SPLINE
SPL {X  -162.820, Y  +428.091, Z    +0.000, E1   +59.583, E3 +218892.152}
SPL {X  -162.820, Y  +410.436, Z    +0.000, E1   +60.611, E3 +218906.354}
SPL {X  -162.820, Y  +392.633, Z    +0.000, E1   +61.698, E3 +218919.086}
SPL {X  -162.753, Y  +375.814, Z    +0.000, E1   +62.427, E3 +218932.608}
SPL {X  -161.572, Y  +360.382, Z    +0.000, E1   +62.315, E3 +218950.211}
SPL {X  -160.005, Y  +350.357, Z    +0.000, E1   +62.043, E3 +218962.774}
SPL {X  -158.606, Y  +343.697, Z    +0.000, E1   +61.897, E3 +218970.997}
SPL {X  -156.311, Y  +334.925, Z    +0.000, E1   +61.505, E3 +218983.343}
SPL {X  -153.198, Y  +325.358, Z    +0.000, E1   +61.117, E3 +218996.036}
SPL {X  -151.022, Y  +319.651, Z    +0.000, E1   +60.776, E3 +219004.208}
SPL {X  -149.105, Y  +315.094, Z    +0.000, E1   +60.301, E3 +219011.961}
SPL {X  -146.196, Y  +308.826, Z    +0.000, E1   +59.961, E3 +219020.668}
SPL {X  -143.704, Y  +303.952, Z    +0.000, E1   +59.374, E3 +219029.025}
SPL {X  -140.940, Y  +298.976, Z    +0.000, E1   +59.075, E3 +219035.950}
SPL {X  -137.763, Y  +293.715, Z    +0.000, E1   +58.761, E3 +219043.057}
SPL {X  -129.725, Y  +282.103, Z    +0.000, E1   +61.069, E3 +219044.560}
SPL {X  -106.695, Y  +257.510, Z    +0.000, E1   +52.408, E3 +219145.282}
SPL {X  -104.122, Y  +255.325, Z    +0.000, E1   +51.312, E3 +219235.340}
ENDSPLINE

SPLINE
SPL {X  -140.007, Y  +297.383, Z    +0.000, E1   +42.766, E3 +219274.665}
SPL {X  -156.919, Y  +337.064, Z    +0.000, E1   +27.647, E3 +219280.816}
SPL {X  -160.736, Y  +354.534, Z    +0.000, E1   +18.553, E3 +219283.511}
SPL {X  -162.078, Y  +364.978, Z    +0.000, E1   +12.369, E3 +219285.196}
SPL {X  -162.656, Y  +373.196, Z    +0.000, E1    +6.960, E3 +219284.692}
SPL {X  -162.819, Y  +379.805, Z    +0.000, E1    +2.285, E3 +219284.816}
SPL {X  -162.820, Y  +382.797, Z    +0.000, E1    -0.206, E3 +219284.322}
SPL {X  -162.820, Y  +386.214, Z    +0.000, E1    -4.241, E3 +219284.088}
SPL {X  -162.820, Y  +390.506, Z    +0.000, E1   -10.770, E3 +219283.854}
SPL {X  -162.820, Y  +394.643, Z    +0.000, E1   -17.317, E3 +219283.808}
SPL {X  -162.820, Y  +401.515, Z    +0.000, E1   -27.960, E3 +219284.628}
SPL {X  -162.820, Y  +412.105, Z    +0.000, E1   -42.847, E3 +219283.620}
SPL {X  -162.820, Y  +422.796, Z    +0.000, E1   -52.392, E3 +219284.841}
SPL {X  -162.820, Y  +474.423, Z    +0.000, E1   -65.078, E3 +219305.892}
SPL {X  -162.820, Y  +578.686, Z    +0.000, E1   -67.085, E3 +219375.056}
ENDSPLINE

SPLINE
SPL {X  -162.820, Y  +565.364, Z    +0.000, E1   -63.589, E3 +219389.056}
ENDSPLINE

SPLINE
SPL {X  -162.820, Y  +574.608, Z    +0.000, E1   -63.370, E3 +219400.315}
SPL {X  -162.820, Y  +584.314, Z    +0.000, E1   -63.342, E3 +219410.607}
SPL {X  -162.820, Y  +593.857, Z    +0.000, E1   -63.382, E3 +219420.310}
SPL {X  -162.820, Y  +602.272, Z    +0.000, E1   -63.279, E3 +219429.838}
SPL {X  -162.820, Y  +613.309, Z    +0.000, E1   -63.489, E3 +219439.836}
SPL {X  -162.820, Y  +627.013, Z    +0.000, E1   -63.389, E3 +219455.057}
SPL {X  -162.820, Y  +642.772, Z    +0.000, E1   -63.348, E3 +219471.716}
SPL {X  -162.820, Y  +651.969, Z    +0.000, E1   -63.137, E3 +219482.778}
SPL {X  -162.820, Y  +662.662, Z    +0.000, E1   -63.383, E3 +219492.236}
SPL {X  -162.819, Y  +673.983, Z    +0.000, E1   -63.398, E3 +219503.958}
SPL {X  -162.399, Y  +685.202, Z    +0.000, E1   -63.235, E3 +219516.952}
SPL {X  -161.289, Y  +695.772, Z    +0.000, E1   -63.167, E3 +219528.402}
SPL {X  -160.212, Y  +702.527, Z    +0.000, E1   -62.898, E3 +219537.383}
SPL {X  -158.647, Y  +710.128, Z    +0.000, E1   -62.776, E3 +219546.206}
SPL {X  -156.957, Y  +716.799, Z    +0.000, E1   -62.460, E3 +219555.324}
SPL {X  -155.130, Y  +722.947, Z    +0.000, E1   -62.207, E3 +219563.436}
SPL {X  -152.287, Y  +731.112, Z    +0.000, E1   -61.798, E3 +219574.711}
SPL {X  -149.420, Y  +738.185, Z    +0.000, E1   -61.282, E3 +219585.120}
SPL {X  -146.033, Y  +745.504, Z    +0.000, E1   -60.844, E3 +219595.387}
SPL {X  -142.518, Y  +752.234, Z    +0.000, E1   -60.144, E3 +219606.013}
SPL {X  -139.430, Y  +757.582, Z    +0.000, E1   -59.554, E3 +219614.545}
SPL {X  -135.510, Y  +763.762, Z    +0.000, E1   -59.735, E3 +219620.066}
SPL {X  -130.418, Y  +770.976, Z    +0.000, E1   -60.870, E3 +219622.223}
SPL {X  -100.103, Y  +801.912, Z    +0.000, E1   -53.794, E3 +219718.546}
ENDSPLINE

SPLINE
SPL {X  -112.938, Y  +790.784, Z    +0.000, E1   -51.983, E3 +219854.068}
SPL {X  -141.567, Y  +753.931, Z    +0.000, E1   -42.659, E3 +219860.676}
SPL {X  -155.442, Y  +721.958, Z    +0.000, E1   -30.769, E3 +219867.583}
SPL {X  -161.417, Y  +694.832, Z    +0.000, E1   -16.464, E3 +219871.551}
SPL {X  -162.719, Y  +679.228, Z    +0.000, E1    -6.085, E3 +219871.875}
SPL {X  -162.820, Y  +673.638, Z    +0.000, E1    -1.806, E3 +219871.665}
SPL {X  -162.820, Y  +671.474, Z    +0.000, E1    -0.022, E3 +219871.261}
SPL {X  -162.820, Y  +668.525, Z    +0.000, E1    +3.543, E3 +219870.955}
SPL {X  -162.820, Y  +663.189, Z    +0.000, E1   +11.952, E3 +219870.944}
SPL {X  -162.820, Y  +655.445, Z    +0.000, E1   +24.952, E3 +219870.890}
SPL {X  -162.820, Y  +644.088, Z    +0.000, E1   +41.840, E3 +219871.026}
SPL {X  -162.820, Y  +632.645, Z    +0.000, E1   +53.114, E3 +219871.762}
SPL {X  -162.820, Y  +584.142, Z    +0.000, E1   +66.966, E3 +219887.104}
SPL {X  -162.820, Y  +471.906, Z    +0.000, E1   +66.781, E3 +219969.346}
SPL {X  -162.820, Y  +470.218, Z    +0.000, E1   +64.979, E3 +219985.346}
SPL {X  -162.820, Y  +452.619, Z    +0.000, E1   +64.912, E3 +220003.024}
SPL {X  -162.820, Y  +437.579, Z    +0.000, E1   +64.893, E3 +220017.707}
SPL {X  -162.820, Y  +425.248, Z    +0.000, E1   +64.950, E3 +220029.294}
SPL {X  -162.820, Y  +417.868, Z    +0.000, E1   +64.478, E3 +220040.113}
ENDSPLINE

SPLINE
SPL {X  -162.820, Y  +442.889, Z    +0.000, E1   +58.918, E3 +220052.293}
ENDSPLINE

SPLINE
SPL {X  -162.820, Y  +428.091, Z    +0.000, E1   +59.583, E3 +220066.065}
SPL {X  -162.820, Y  +410.436, Z    +0.000, E1   +60.611, E3 +220080.267}
SPL {X  -162.820, Y  +392.633, Z    +0.000, E1   +61.698, E3 +220092.999}
SPL {X  -162.753, Y  +375.814, Z    +0.000, E1   +62.427, E3 +220106.521}
SPL {X  -161.572, Y  +360.382, Z    +0.000, E1   +62.315, E3 +220124.124}
SPL {X  -160.005, Y  +350.357, Z    +0.000, E1   +62.043, E3 +220136.687}
SPL {X  -158.606, Y  +343.697, Z    +0.000, E1   +61.897, E3 +220144.910}
SPL {X  -156.311, Y  +334.925, Z    +0.000, E1   +61.505, E3 +220157.256}
SPL {X  -153.198, Y  +325.358, Z    +0.000, E1   +61.117, E3 +220169.949}
SPL {X  -151.022, Y  +319.651, Z    +0.000, E1   +60.776, E3 +220178.121}
SPL {X  -149.105, Y  +315.094, Z    +0.000, E1   +60.301, E3 +220185.874}
SPL {X  -146.196, Y  +308.826, Z    +0.000, E1   +59.961, E3 +220194.581}
SPL {X  -143.704, Y  +303.952, Z    +0.000, E1   +59.374, E3 +220202.938}
SPL {X  -140.940, Y  +298.976, Z    +0.000, E1   +59.075, E3 +220209.863}
SPL {X  -137.763, Y  +293.715, Z    +0.000, E1   +58.761, E3 +220216.970}
SPL {X  -129.725, Y  +282.103, Z    +0.000, E1   +61.069, E3 +220218.473}
SPL {X  -106.695, Y  +257.510, Z    +0.000, E1   +52.408, E3 +220319.195}
SPL {X  -104.122, Y  +255.325, Z    +0.000, E1   +51.312, E3 +220409.253}
ENDSPLINE

SPLINE
SPL {X  -140.007, Y  +297.383, Z    +0.000, E1   +42.766, E3 +220448.578}
SPL {X  -155.551, Y  +332.393, Z    +0.000, E1   +29.794, E3 +220454.500}
SPL {X  -159.755, Y  +349.054, Z    +0.000, E1   +21.610, E3 +220456.372}
SPL {X  -162.078, Y  +364.978, Z    +0.000, E1   +12.369, E3 +220459.109}
SPL {X  -162.752, Y  +375.778, Z    +0.000, E1    +5.236, E3 +220458.818}
SPL {X  -162.820, Y  +381.939, Z    +0.000, E1    +0.593, E3 +220458.446}
SPL {X  -162.820, Y  +383.993, Z    +0.000, E1    -1.497, E3 +220458.019}
SPL {X  -162.820, Y  +388.628, Z    +0.000, E1    -7.678, E3 +220457.921}
SPL {X  -162.820, Y  +394.643, Z    +0.000, E1   -17.317, E3 +220457.721}
SPL {X  -162.820, Y  +401.515, Z    +0.000, E1   -27.960, E3 +220458.541}
SPL {X  -162.820, Y  +412.105, Z    +0.000, E1   -42.847, E3 +220457.533}
SPL {X  -162.820, Y  +422.796, Z    +0.000, E1   -52.392, E3 +220458.754}
SPL {X  -162.820, Y  +474.423, Z    +0.000, E1   -65.078, E3 +220479.805}
SPL {X  -162.820, Y  +578.686, Z    +0.000, E1   -67.085, E3 +220548.969}
ENDSPLINE

SPLINE
SPL {X  -162.820, Y  +565.364, Z    +0.000, E1   -63.589, E3 +220562.969}
ENDSPLINE

SPLINE
SPL {X  -162.820, Y  +574.608, Z    +0.000, E1   -63.370, E3 +220574.228}
SPL {X  -162.820, Y  +584.314, Z    +0.000, E1   -63.342, E3 +220584.520}
SPL {X  -162.820, Y  +593.857, Z    +0.000, E1   -63.382, E3 +220594.223}
SPL {X  -162.820, Y  +602.272, Z    +0.000, E1   -63.279, E3 +220603.751}
SPL {X  -162.820, Y  +613.309, Z    +0.000, E1   -63.489, E3 +220613.749}
SPL {X  -162.820, Y  +627.013, Z    +0.000, E1   -63.389, E3 +220628.970}
SPL {X  -162.820, Y  +642.772, Z    +0.000, E1   -63.348, E3 +220645.629}
SPL {X  -162.820, Y  +651.969, Z    +0.000, E1   -63.137, E3 +220656.691}
SPL {X  -162.820, Y  +662.662, Z    +0.000, E1   -63.383, E3 +220666.149}
SPL {X  -162.819, Y  +673.983, Z    +0.000, E1   -63.398, E3 +220677.871}
SPL {X  -162.399, Y  +685.202, Z    +0.000, E1   -63.235, E3 +220690.865}
SPL {X  -161.289, Y  +695.772, Z    +0.000, E1   -63.167, E3 +220702.315}
SPL {X  -160.212, Y  +702.527, Z    +0.000, E1   -62.898, E3 +220711.296}
SPL {X  -158.647, Y  +710.128, Z    +0.000, E1   -62.776, E3 +220720.119}
SPL {X  -156.957, Y  +716.799, Z    +0.000, E1   -62.460, E3 +220729.237}
SPL {X  -154.447, Y  +725.041, Z    +0.000, E1   -62.170, E3 +220739.894}
SPL {X  -151.721, Y  +732.586, Z    +0.000, E1   -61.616, E3 +220751.144}
SPL {X  -149.420, Y  +738.185, Z    +0.000, E1   -61.282, E3 +220759.033}
SPL {X  -146.033, Y  +745.504, Z    +0.000, E1   -60.844, E3 +220769.300}
SPL {X  -142.518, Y  +752.234, Z    +0.000, E1   -60.144, E3 +220779.926}
SPL {X  -139.430, Y  +757.582, Z    +0.000, E1   -59.554, E3 +220788.458}
SPL {X  -135.510, Y  +763.762, Z    +0.000, E1   -59.735, E3 +220793.979}
SPL {X  -130.418, Y  +770.976, Z    +0.000, E1   -60.870, E3 +220796.136}
SPL {X  -100.103, Y  +801.912, Z    +0.000, E1   -53.794, E3 +220892.459}
ENDSPLINE

SPLINE
SPL {X  -112.938, Y  +790.784, Z    +0.000, E1   -51.983, E3 +221027.981}
SPL {X  -141.567, Y  +753.931, Z    +0.000, E1   -42.659, E3 +221034.589}
SPL {X  -155.442, Y  +721.958, Z    +0.000, E1   -30.769, E3 +221041.496}
SPL {X  -160.289, Y  +702.098, Z    +0.000, E1   -20.686, E3 +221045.224}
SPL {X  -162.312, Y  +686.349, Z    +0.000, E1   -11.031, E3 +221045.630}
SPL {X  -162.811, Y  +675.182, Z    +0.000, E1    -3.078, E3 +221045.704}
SPL {X  -162.820, Y  +671.474, Z    +0.000, E1    -0.022, E3 +221045.174}
SPL {X  -162.820, Y  +668.525, Z    +0.000, E1    +3.543, E3 +221044.868}
SPL {X  -162.820, Y  +663.189, Z    +0.000, E1   +11.952, E3 +221044.857}
SPL {X  -162.820, Y  +655.445, Z    +0.000, E1   +24.952, E3 +221044.803}
SPL {X  -162.820, Y  +644.088, Z    +0.000, E1   +41.840, E3 +221044.939}
SPL {X  -162.820, Y  +632.645, Z    +0.000, E1   +53.114, E3 +221045.675}
SPL {X  -162.820, Y  +584.142, Z    +0.000, E1   +66.966, E3 +221061.017}
SPL {X  -162.820, Y  +471.906, Z    +0.000, E1   +66.781, E3 +221143.259}
SPL {X  -162.820, Y  +470.218, Z    +0.000, E1   +64.979, E3 +221159.259}
SPL {X  -162.820, Y  +452.619, Z    +0.000, E1   +64.912, E3 +221176.937}
SPL {X  -162.820, Y  +437.579, Z    +0.000, E1   +64.893, E3 +221191.620}
SPL {X  -162.820, Y  +425.248, Z    +0.000, E1   +64.950, E3 +221203.207}
SPL {X  -162.820, Y  +417.868, Z    +0.000, E1   +64.478, E3 +221214.026}
ENDSPLINE

SPLINE
SPL {X  -162.820, Y  +442.889, Z    +0.000, E1   +58.918, E3 +221226.206}
ENDSPLINE

SPLINE
SPL {X  -162.820, Y  +428.091, Z    +0.000, E1   +59.583, E3 +221239.978}
SPL {X  -162.820, Y  +410.436, Z    +0.000, E1   +60.611, E3 +221254.180}
SPL {X  -162.820, Y  +392.633, Z    +0.000, E1   +61.698, E3 +221266.912}
SPL {X  -162.753, Y  +375.814, Z    +0.000, E1   +62.427, E3 +221280.434}
SPL {X  -161.572, Y  +360.382, Z    +0.000, E1   +62.315, E3 +221298.037}
SPL {X  -160.005, Y  +350.357, Z    +0.000, E1   +62.043, E3 +221310.600}
SPL {X  -157.973, Y  +341.066, Z    +0.000, E1   +61.800, E3 +221322.517}
SPL {X  -155.627, Y  +332.640, Z    +0.000, E1   +61.354, E3 +221334.432}
SPL {X  -153.198, Y  +325.358, Z    +0.000, E1   +61.117, E3 +221343.862}
SPL {X  -151.022, Y  +319.651, Z    +0.000, E1   +60.776, E3 +221352.034}
SPL {X  -149.105, Y  +315.094, Z    +0.000, E1   +60.301, E3 +221359.787}
SPL {X  -146.196, Y  +308.826, Z    +0.000, E1   +59.961, E3 +221368.494}
SPL {X  -143.704, Y  +303.952, Z    +0.000, E1   +59.374, E3 +221376.851}
SPL {X  -140.940, Y  +298.976, Z    +0.000, E1   +59.075, E3 +221383.776}
SPL {X  -137.763, Y  +293.715, Z    +0.000, E1   +58.761, E3 +221390.883}
SPL {X  -129.725, Y  +282.103, Z    +0.000, E1   +61.069, E3 +221392.386}
SPL {X  -106.695, Y  +257.510, Z    +0.000, E1   +52.408, E3 +221493.108}
SPL {X  -104.122, Y  +255.325, Z    +0.000, E1   +51.312, E3 +221583.166}
ENDSPLINE

SPLINE
SPL {X  -140.007, Y  +297.383, Z    +0.000, E1   +42.766, E3 +221622.491}
SPL {X  -156.919, Y  +337.064, Z    +0.000, E1   +27.647, E3 +221628.642}
SPL {X  -161.737, Y  +361.753, Z    +0.000, E1   +14.421, E3 +221632.539}
SPL {X  -162.752, Y  +375.778, Z    +0.000, E1    +5.236, E3 +221632.731}
SPL {X  -162.820, Y  +380.849, Z    +0.000, E1    +1.416, E3 +221632.495}
SPL {X  -162.820, Y  +383.416, Z    +0.000, E1    -0.722, E3 +221632.066}
SPL {X  -162.820, Y  +388.628, Z    +0.000, E1    -7.678, E3 +221631.834}
SPL {X  -162.820, Y  +394.643, Z    +0.000, E1   -17.317, E3 +221631.634}
SPL {X  -162.820, Y  +401.515, Z    +0.000, E1   -27.960, E3 +221632.454}
SPL {X  -162.820, Y  +412.105, Z    +0.000, E1   -42.847, E3 +221631.447}
SPL {X  -162.820, Y  +422.796, Z    +0.000, E1   -52.392, E3 +221632.667}
SPL {X  -162.820, Y  +474.423, Z    +0.000, E1   -65.078, E3 +221653.718}
SPL {X  -162.820, Y  +578.686, Z    +0.000, E1   -67.085, E3 +221722.883}
ENDSPLINE

SPLINE
SPL {X  -162.820, Y  +565.364, Z    +0.000, E1   -63.589, E3 +221736.883}
ENDSPLINE

SPLINE
SPL {X  -162.820, Y  +574.608, Z    +0.000, E1   -63.370, E3 +221748.141}
SPL {X  -162.820, Y  +584.314, Z    +0.000, E1   -63.342, E3 +221758.433}
SPL {X  -162.820, Y  +593.857, Z    +0.000, E1   -63.382, E3 +221768.136}
SPL {X  -162.820, Y  +602.272, Z    +0.000, E1   -63.279, E3 +221777.664}
SPL {X  -162.820, Y  +613.309, Z    +0.000, E1   -63.489, E3 +221787.662}
SPL {X  -162.820, Y  +619.956, Z    +0.000, E1   -63.110, E3 +221797.349}
SPL {X  -162.820, Y  +634.513, Z    +0.000, E1   -63.471, E3 +221810.115}
SPL {X  -162.820, Y  +648.936, Z    +0.000, E1   -63.278, E3 +221826.570}
SPL {X  -162.820, Y  +662.662, Z    +0.000, E1   -63.383, E3 +221840.062}
SPL {X  -162.819, Y  +673.983, Z    +0.000, E1   -63.398, E3 +221851.785}
SPL {X  -162.399, Y  +685.202, Z    +0.000, E1   -63.235, E3 +221864.778}
SPL {X  -161.289, Y  +695.772, Z    +0.000, E1   -63.167, E3 +221876.228}
SPL {X  -160.212, Y  +702.527, Z    +0.000, E1   -62.898, E3 +221885.209}
SPL {X  -158.647, Y  +710.128, Z    +0.000, E1   -62.776, E3 +221894.032}
SPL {X  -156.957, Y  +716.799, Z    +0.000, E1   -62.460, E3 +221903.150}
SPL {X  -154.447, Y  +725.041, Z    +0.000, E1   -62.170, E3 +221913.807}
SPL {X  -151.721, Y  +732.586, Z    +0.000, E1   -61.616, E3 +221925.057}
SPL {X  -149.420, Y  +738.185, Z    +0.000, E1   -61.282, E3 +221932.946}
SPL {X  -146.033, Y  +745.504, Z    +0.000, E1   -60.844, E3 +221943.213}
SPL {X  -142.518, Y  +752.234, Z    +0.000, E1   -60.144, E3 +221953.839}
SPL {X  -139.430, Y  +757.582, Z    +0.000, E1   -59.554, E3 +221962.371}
SPL {X  -134.550, Y  +765.187, Z    +0.000, E1   -59.954, E3 +221968.322}
SPL {X  -100.103, Y  +801.912, Z    +0.000, E1   -53.794, E3 +222066.372}
ENDSPLINE

SPLINE
SPL {X  -112.938, Y  +790.784, Z    +0.000, E1   -51.983, E3 +222201.894}
SPL {X  -145.058, Y  +747.450, Z    +0.000, E1   -40.634, E3 +222210.004}
SPL {X  -158.857, Y  +709.206, Z    +0.000, E1   -24.633, E3 +222217.973}
SPL {X  -161.919, Y  +690.607, Z    +0.000, E1   -13.733, E3 +222219.453}
SPL {X  -162.719, Y  +679.228, Z    +0.000, E1    -6.085, E3 +222219.702}
SPL {X  -162.820, Y  +673.638, Z    +0.000, E1    -1.806, E3 +222219.491}
SPL {X  -162.820, Y  +671.474, Z    +0.000, E1    -0.022, E3 +222219.087}
SPL {X  -162.820, Y  +668.525, Z    +0.000, E1    +3.543, E3 +222218.781}
SPL {X  -162.820, Y  +663.189, Z    +0.000, E1   +11.952, E3 +222218.770}
SPL {X  -162.820, Y  +655.445, Z    +0.000, E1   +24.952, E3 +222218.716}
SPL {X  -162.820, Y  +644.088, Z    +0.000, E1   +41.840, E3 +222218.852}
SPL {X  -162.820, Y  +632.645, Z    +0.000, E1   +53.114, E3 +222219.588}
SPL {X  -162.820, Y  +584.142, Z    +0.000, E1   +66.966, E3 +222234.931}
SPL {X  -162.820, Y  +471.906, Z    +0.000, E1   +66.781, E3 +222317.172}
SPL {X  -162.820, Y  +470.218, Z    +0.000, E1   +64.979, E3 +222333.172}
SPL {X  -162.820, Y  +452.619, Z    +0.000, E1   +64.912, E3 +222350.850}
SPL {X  -162.820, Y  +437.579, Z    +0.000, E1   +64.893, E3 +222365.533}
SPL {X  -162.820, Y  +425.248, Z    +0.000, E1   +64.950, E3 +222377.120}
SPL {X  -162.820, Y  +417.868, Z    +0.000, E1   +64.478, E3 +222387.939}
ENDSPLINE

SPLINE
SPL {X  -162.820, Y  +442.889, Z    +0.000, E1   +58.918, E3 +222400.119}
ENDSPLINE

SPLINE
SPL {X  -162.820, Y  +428.091, Z    +0.000, E1   +59.583, E3 +222413.891}
SPL {X  -162.820, Y  +417.107, Z    +0.000, E1   +60.148, E3 +222423.293}
SPL {X  -162.820, Y  +398.797, Z    +0.000, E1   +61.348, E3 +222436.425}
SPL {X  -162.753, Y  +375.814, Z    +0.000, E1   +62.427, E3 +222454.347}
SPL {X  -161.572, Y  +360.382, Z    +0.000, E1   +62.315, E3 +222471.950}
SPL {X  -160.005, Y  +350.357, Z    +0.000, E1   +62.043, E3 +222484.513}
SPL {X  -158.606, Y  +343.697, Z    +0.000, E1   +61.897, E3 +222492.736}
SPL {X  -156.311, Y  +334.925, Z    +0.000, E1   +61.505, E3 +222505.082}
SPL {X  -153.198, Y  +325.358, Z    +0.000, E1   +61.117, E3 +222517.775}
SPL {X  -151.022, Y  +319.651, Z    +0.000, E1   +60.776, E3 +222525.947}
SPL {X  -149.105, Y  +315.094, Z    +0.000, E1   +60.301, E3 +222533.700}
SPL {X  -146.196, Y  +308.826, Z    +0.000, E1   +59.961, E3 +222542.407}
SPL {X  -143.704, Y  +303.952, Z    +0.000, E1   +59.374, E3 +222550.764}
SPL {X  -140.940, Y  +298.976, Z    +0.000, E1   +59.075, E3 +222557.689}
SPL {X  -137.763, Y  +293.715, Z    +0.000, E1   +58.761, E3 +222564.796}
SPL {X  -129.725, Y  +282.103, Z    +0.000, E1   +61.069, E3 +222566.299}
SPL {X  -106.695, Y  +257.510, Z    +0.000, E1   +52.408, E3 +222667.021}
SPL {X  -104.122, Y  +255.325, Z    +0.000, E1   +51.312, E3 +222757.079}
ENDSPLINE

SPLINE
SPL {X  -140.007, Y  +297.383, Z    +0.000, E1   +42.766, E3 +222796.404}
SPL {X  -156.919, Y  +337.064, Z    +0.000, E1   +27.647, E3 +222802.555}
SPL {X  -160.736, Y  +354.534, Z    +0.000, E1   +18.553, E3 +222805.250}
SPL {X  -162.078, Y  +364.978, Z    +0.000, E1   +12.369, E3 +222806.936}
SPL {X  -162.656, Y  +373.196, Z    +0.000, E1    +6.960, E3 +222806.431}
SPL {X  -162.819, Y  +379.805, Z    +0.000, E1    +2.285, E3 +222806.555}
SPL {X  -162.820, Y  +383.416, Z    +0.000, E1    -0.722, E3 +222805.979}
SPL {X  -162.820, Y  +388.628, Z    +0.000, E1    -7.678, E3 +222805.747}
SPL {X  -162.820, Y  +394.643, Z    +0.000, E1   -17.317, E3 +222805.547}
SPL {X  -162.820, Y  +401.515, Z    +0.000, E1   -27.960, E3 +222806.367}
SPL {X  -162.820, Y  +412.105, Z    +0.000, E1   -42.847, E3 +222805.360}
SPL {X  -162.820, Y  +422.796, Z    +0.000, E1   -52.392, E3 +222806.580}
SPL {X  -162.820, Y  +474.423, Z    +0.000, E1   -65.078, E3 +222827.631}
SPL {X  -162.820, Y  +578.686, Z    +0.000, E1   -67.085, E3 +222896.796}
ENDSPLINE

SPLINE
SPL {X  -162.820, Y  +565.364, Z    +0.000, E1   -63.589, E3 +222910.796}
ENDSPLINE

SPLINE
SPL {X  -162.820, Y  +574.608, Z    +0.000, E1   -63.370, E3 +222922.054}
SPL {X  -162.820, Y  +584.314, Z    +0.000, E1   -63.342, E3 +222932.346}
SPL {X  -162.820, Y  +593.857, Z    +0.000, E1   -63.382, E3 +222942.049}
SPL {X  -162.820, Y  +602.272, Z    +0.000, E1   -63.279, E3 +222951.577}
SPL {X  -162.820, Y  +613.309, Z    +0.000, E1   -63.489, E3 +222961.575}
SPL {X  -162.820, Y  +619.956, Z    +0.000, E1   -63.110, E3 +222971.262}
SPL {X  -162.820, Y  +631.846, Z    +0.000, E1   -63.529, E3 +222980.652}
SPL {X  -162.820, Y  +642.772, Z    +0.000, E1   -63.348, E3 +222993.455}
SPL {X  -162.820, Y  +658.642, Z    +0.000, E1   -63.324, E3 +223010.370}
SPL {X  -162.819, Y  +673.983, Z    +0.000, E1   -63.398, E3 +223025.698}
SPL {X  -162.399, Y  +685.202, Z    +0.000, E1   -63.235, E3 +223038.691}
SPL {X  -161.289, Y  +695.772, Z    +0.000, E1   -63.167, E3 +223050.141}
SPL {X  -160.212, Y  +702.527, Z    +0.000, E1   -62.898, E3 +223059.122}
SPL {X  -158.647, Y  +710.128, Z    +0.000, E1   -62.776, E3 +223067.945}
SPL {X  -156.957, Y  +716.799, Z    +0.000, E1   -62.460, E3 +223077.063}
SPL {X  -154.447, Y  +725.041, Z    +0.000, E1   -62.170, E3 +223087.720}
SPL {X  -151.721, Y  +732.586, Z    +0.000, E1   -61.616, E3 +223098.970}
SPL {X  -149.420, Y  +738.185, Z    +0.000, E1   -61.282, E3 +223106.859}
SPL {X  -146.033, Y  +745.504, Z    +0.000, E1   -60.844, E3 +223117.126}
SPL {X  -142.518, Y  +752.234, Z    +0.000, E1   -60.144, E3 +223127.752}
SPL {X  -139.430, Y  +757.582, Z    +0.000, E1   -59.554, E3 +223136.284}
SPL {X  -134.550, Y  +765.187, Z    +0.000, E1   -59.954, E3 +223142.236}
SPL {X  -100.103, Y  +801.912, Z    +0.000, E1   -53.794, E3 +223240.285}
ENDSPLINE

SPLINE
SPL {X  -112.938, Y  +790.784, Z    +0.000, E1   -51.983, E3 +223375.807}
SPL {X  -141.567, Y  +753.931, Z    +0.000, E1   -42.659, E3 +223382.415}
SPL {X  -155.442, Y  +721.958, Z    +0.000, E1   -30.769, E3 +223389.322}
SPL {X  -161.417, Y  +694.832, Z    +0.000, E1   -16.464, E3 +223393.291}
SPL {X  -162.719, Y  +679.228, Z    +0.000, E1    -6.085, E3 +223393.615}
SPL {X  -162.820, Y  +673.638, Z    +0.000, E1    -1.806, E3 +223393.404}
SPL {X  -162.820, Y  +671.474, Z    +0.000, E1    -0.022, E3 +223393.000}
SPL {X  -162.820, Y  +668.525, Z    +0.000, E1    +3.543, E3 +223392.694}
SPL {X  -162.820, Y  +663.189, Z    +0.000, E1   +11.952, E3 +223392.683}
SPL {X  -162.820, Y  +655.445, Z    +0.000, E1   +24.952, E3 +223392.629}
SPL {X  -162.820, Y  +644.088, Z    +0.000, E1   +41.840, E3 +223392.765}
SPL {X  -162.820, Y  +632.645, Z    +0.000, E1   +53.114, E3 +223393.501}
SPL {X  -162.820, Y  +584.142, Z    +0.000, E1   +66.966, E3 +223408.844}
SPL {X  -162.820, Y  +471.906, Z    +0.000, E1   +66.781, E3 +223491.085}
SPL {X  -162.820, Y  +470.218, Z    +0.000, E1   +64.979, E3 +223507.085}
SPL {X  -162.820, Y  +452.619, Z    +0.000, E1   +64.912, E3 +223524.763}
SPL {X  -162.820, Y  +437.579, Z    +0.000, E1   +64.893, E3 +223539.446}
SPL {X  -162.820, Y  +425.248, Z    +0.000, E1   +64.950, E3 +223551.033}
SPL {X  -162.820, Y  +417.868, Z    +0.000, E1   +64.478, E3 +223561.852}
ENDSPLINE

SPLINE
SPL {X  -162.820, Y  +447.149, Z    +0.000, E1   +58.721, E3 +223569.848}
ENDSPLINE

SPLINE
SPL {X  -162.820, Y  +431.862, Z    +0.000, E1   +59.419, E3 +223584.395}
SPL {X  -162.820, Y  +417.107, Z    +0.000, E1   +60.148, E3 +223597.206}
SPL {X  -162.820, Y  +398.797, Z    +0.000, E1   +61.348, E3 +223610.338}
SPL {X  -162.819, Y  +379.881, Z    +0.000, E1   +62.356, E3 +223624.168}
SPL {X  -162.597, Y  +371.985, Z    +0.000, E1   +62.420, E3 +223632.292}
SPL {X  -161.953, Y  +363.716, Z    +0.000, E1   +62.355, E3 +223641.749}
SPL {X  -160.528, Y  +353.277, Z    +0.000, E1   +62.144, E3 +223654.745}
SPL {X  -158.606, Y  +343.697, Z    +0.000, E1   +61.897, E3 +223666.649}
SPL {X  -156.311, Y  +334.925, Z    +0.000, E1   +61.505, E3 +223678.995}
SPL {X  -153.198, Y  +325.358, Z    +0.000, E1   +61.117, E3 +223691.688}
SPL {X  -151.022, Y  +319.651, Z    +0.000, E1   +60.776, E3 +223699.861}
SPL {X  -149.105, Y  +315.094, Z    +0.000, E1   +60.301, E3 +223707.614}
SPL {X  -146.196, Y  +308.826, Z    +0.000, E1   +59.961, E3 +223716.320}
SPL {X  -143.704, Y  +303.952, Z    +0.000, E1   +59.374, E3 +223724.677}
SPL {X  -140.940, Y  +298.976, Z    +0.000, E1   +59.075, E3 +223731.602}
SPL {X  -137.763, Y  +293.715, Z    +0.000, E1   +58.761, E3 +223738.709}
SPL {X  -129.725, Y  +282.103, Z    +0.000, E1   +61.069, E3 +223740.212}
SPL {X  -106.695, Y  +257.510, Z    +0.000, E1   +52.408, E3 +223840.935}
SPL {X  -104.122, Y  +255.325, Z    +0.000, E1   +51.312, E3 +223930.992}
ENDSPLINE

SPLINE
SPL {X  -140.007, Y  +297.383, Z    +0.000, E1   +42.766, E3 +223970.317}
SPL {X  -155.551, Y  +332.393, Z    +0.000, E1   +29.794, E3 +223976.239}
SPL {X  -159.755, Y  +349.054, Z    +0.000, E1   +21.610, E3 +223978.112}
SPL {X  -162.078, Y  +364.978, Z    +0.000, E1   +12.369, E3 +223980.849}
SPL {X  -162.752, Y  +375.778, Z    +0.000, E1    +5.236, E3 +223980.557}
SPL {X  -162.820, Y  +382.443, Z    +0.000, E1    +0.212, E3 +223980.037}
SPL {X  -162.820, Y  +386.214, Z    +0.000, E1    -4.241, E3 +223979.740}
SPL {X  -162.820, Y  +390.506, Z    +0.000, E1   -10.770, E3 +223979.507}
SPL {X  -162.820, Y  +394.643, Z    +0.000, E1   -17.317, E3 +223979.460}
SPL {X  -162.820, Y  +401.515, Z    +0.000, E1   -27.960, E3 +223980.281}
SPL {X  -162.820, Y  +412.105, Z    +0.000, E1   -42.847, E3 +223979.273}
SPL {X  -162.820, Y  +422.796, Z    +0.000, E1   -52.392, E3 +223980.493}
SPL {X  -162.820, Y  +474.423, Z    +0.000, E1   -65.078, E3 +224001.544}
SPL {X  -162.820, Y  +578.686, Z    +0.000, E1   -67.085, E3 +224070.709}
ENDSPLINE

SPLINE
SPL {X  -162.820, Y  +565.364, Z    +0.000, E1   -63.589, E3 +224084.709}
ENDSPLINE

SPLINE
SPL {X  -162.820, Y  +574.608, Z    +0.000, E1   -63.370, E3 +224095.967}
SPL {X  -162.820, Y  +584.314, Z    +0.000, E1   -63.342, E3 +224106.259}
SPL {X  -162.820, Y  +593.857, Z    +0.000, E1   -63.382, E3 +224115.962}
SPL {X  -162.820, Y  +602.272, Z    +0.000, E1   -63.279, E3 +224125.490}
SPL {X  -162.820, Y  +613.309, Z    +0.000, E1   -63.489, E3 +224135.488}
SPL {X  -162.820, Y  +627.013, Z    +0.000, E1   -63.389, E3 +224150.709}
SPL {X  -162.820, Y  +642.772, Z    +0.000, E1   -63.348, E3 +224167.368}
SPL {X  -162.820, Y  +658.642, Z    +0.000, E1   -63.324, E3 +224184.283}
SPL {X  -162.819, Y  +673.983, Z    +0.000, E1   -63.398, E3 +224199.611}
SPL {X  -162.617, Y  +681.634, Z    +0.000, E1   -63.169, E3 +224209.233}
SPL {X  -161.618, Y  +693.246, Z    +0.000, E1   -63.233, E3 +224221.090}
SPL {X  -160.212, Y  +702.527, Z    +0.000, E1   -62.898, E3 +224233.035}
SPL {X  -158.647, Y  +710.128, Z    +0.000, E1   -62.776, E3 +224241.858}
SPL {X  -156.957, Y  +716.799, Z    +0.000, E1   -62.460, E3 +224250.976}
SPL {X  -155.130, Y  +722.947, Z    +0.000, E1   -62.207, E3 +224259.088}
SPL {X  -152.287, Y  +731.112, Z    +0.000, E1   -61.798, E3 +224270.363}
SPL {X  -149.420, Y  +738.185, Z    +0.000, E1   -61.282, E3 +224280.772}
SPL {X  -146.033, Y  +745.504, Z    +0.000, E1   -60.844, E3 +224291.039}
SPL {X  -142.518, Y  +752.234, Z    +0.000, E1   -60.144, E3 +224301.666}
SPL {X  -139.430, Y  +757.582, Z    +0.000, E1   -59.554, E3 +224310.197}
SPL {X  -134.550, Y  +765.187, Z    +0.000, E1   -59.954, E3 +224316.149}
SPL {X  -100.103, Y  +801.912, Z    +0.000, E1   -53.794, E3 +224414.198}
ENDSPLINE

SPLINE
SPL {X  -112.938, Y  +790.784, Z    +0.000, E1   -51.983, E3 +224549.720}
SPL {X  -145.058, Y  +747.450, Z    +0.000, E1   -40.634, E3 +224557.830}
SPL {X  -158.857, Y  +709.206, Z    +0.000, E1   -24.633, E3 +224565.799}
SPL {X  -162.312, Y  +686.349, Z    +0.000, E1   -11.031, E3 +224567.369}
SPL {X  -162.811, Y  +675.182, Z    +0.000, E1    -3.078, E3 +224567.443}
SPL {X  -162.820, Y  +670.948, Z    +0.000, E1    +0.412, E3 +224566.842}
SPL {X  -162.820, Y  +667.375, Z    +0.000, E1    +5.386, E3 +224566.531}
SPL {X  -162.820, Y  +663.189, Z    +0.000, E1   +11.952, E3 +224566.596}
SPL {X  -162.820, Y  +657.986, Z    +0.000, E1   +20.997, E3 +224566.309}
SPL {X  -162.820, Y  +650.033, Z    +0.000, E1   +33.465, E3 +224566.779}
SPL {X  -162.820, Y  +635.632, Z    +0.000, E1   +50.654, E3 +224567.104}
SPL {X  -162.820, Y  +584.142, Z    +0.000, E1   +66.966, E3 +224582.757}
SPL {X  -162.820, Y  +466.182, Z    +0.000, E1   +68.456, E3 +224656.527}
ENDSPLINE

SPLINE
SPL {X  -162.820, Y  +475.083, Z    +0.000, E1   +65.244, E3 +224674.228}
ENDSPLINE

SPLINE
SPL {X  -162.820, Y  +465.389, Z    +0.000, E1   +65.015, E3 +224685.245}
SPL {X  -162.820, Y  +452.619, Z    +0.000, E1   +64.912, E3 +224698.677}
SPL {X  -162.820, Y  +437.579, Z    +0.000, E1   +64.893, E3 +224713.359}
SPL {X  -162.820, Y  +425.248, Z    +0.000, E1   +64.950, E3 +224724.946}
SPL {X  -162.820, Y  +417.868, Z    +0.000, E1   +64.478, E3 +224735.765}
ENDSPLINE

SPLINE
SPL {X  -162.820, Y  +442.889, Z    +0.000, E1   +58.918, E3 +224747.945}
ENDSPLINE

SPLINE
SPL {X  -162.820, Y  +428.091, Z    +0.000, E1   +59.583, E3 +224761.717}
SPL {X  -162.820, Y  +417.107, Z    +0.000, E1   +60.148, E3 +224771.119}
SPL {X  -162.820, Y  +398.797, Z    +0.000, E1   +61.348, E3 +224784.251}
SPL {X  -162.819, Y  +379.860, Z    +0.000, E1   +62.359, E3 +224798.081}
SPL {X  -162.598, Y  +372.005, Z    +0.000, E1   +62.416, E3 +224806.205}
SPL {X  -161.953, Y  +363.716, Z    +0.000, E1   +62.355, E3 +224815.662}
SPL {X  -160.528, Y  +353.277, Z    +0.000, E1   +62.144, E3 +224828.658}
SPL {X  -157.973, Y  +341.066, Z    +0.000, E1   +61.800, E3 +224844.256}
SPL {X  -155.627, Y  +332.640, Z    +0.000, E1   +61.354, E3 +224856.171}
SPL {X  -153.198, Y  +325.358, Z    +0.000, E1   +61.117, E3 +224865.601}
SPL {X  -151.022, Y  +319.651, Z    +0.000, E1   +60.776, E3 +224873.774}
SPL {X  -149.105, Y  +315.094, Z    +0.000, E1   +60.301, E3 +224881.527}
SPL {X  -146.196, Y  +308.826, Z    +0.000, E1   +59.961, E3 +224890.233}
SPL {X  -143.704, Y  +303.952, Z    +0.000, E1   +59.374, E3 +224898.590}
SPL {X  -140.940, Y  +298.976, Z    +0.000, E1   +59.075, E3 +224905.515}
SPL {X  -137.763, Y  +293.715, Z    +0.000, E1   +58.761, E3 +224912.622}
SPL {X  -129.725, Y  +282.103, Z    +0.000, E1   +61.069, E3 +224914.125}
SPL {X  -106.695, Y  +257.510, Z    +0.000, E1   +52.408, E3 +225014.848}
SPL {X  -104.122, Y  +255.325, Z    +0.000, E1   +51.312, E3 +225104.905}
ENDSPLINE

SPLINE
SPL {X  -140.007, Y  +297.383, Z    +0.000, E1   +42.766, E3 +225144.230}
SPL {X  -155.551, Y  +332.393, Z    +0.000, E1   +29.794, E3 +225150.152}
SPL {X  -159.755, Y  +349.054, Z    +0.000, E1   +21.610, E3 +225152.025}
SPL {X  -162.078, Y  +364.978, Z    +0.000, E1   +12.369, E3 +225154.762}
SPL {X  -162.752, Y  +375.778, Z    +0.000, E1    +5.236, E3 +225154.470}
SPL {X  -162.820, Y  +382.443, Z    +0.000, E1    +0.212, E3 +225153.950}
SPL {X  -162.820, Y  +386.214, Z    +0.000, E1    -4.241, E3 +225153.653}
SPL {X  -162.820, Y  +390.506, Z    +0.000, E1   -10.770, E3 +225153.420}
SPL {X  -162.820, Y  +394.643, Z    +0.000, E1   -17.317, E3 +225153.373}
SPL {X  -162.820, Y  +401.515, Z    +0.000, E1   -27.960, E3 +225154.194}
SPL {X  -162.820, Y  +412.105, Z    +0.000, E1   -42.847, E3 +225153.186}
SPL {X  -162.820, Y  +422.796, Z    +0.000, E1   -52.392, E3 +225154.406}
SPL {X  -162.820, Y  +474.423, Z    +0.000, E1   -65.078, E3 +225175.457}
SPL {X  -162.820, Y  +578.686, Z    +0.000, E1   -67.085, E3 +225244.622}
ENDSPLINE

SPLINE
SPL {X  -162.820, Y  +565.364, Z    +0.000, E1   -63.589, E3 +225258.622}
ENDSPLINE

SPLINE
SPL {X  -162.820, Y  +574.608, Z    +0.000, E1   -63.370, E3 +225269.880}
SPL {X  -162.820, Y  +584.314, Z    +0.000, E1   -63.342, E3 +225280.172}
SPL {X  -162.820, Y  +593.857, Z    +0.000, E1   -63.382, E3 +225289.875}
SPL {X  -162.820, Y  +602.272, Z    +0.000, E1   -63.279, E3 +225299.403}
SPL {X  -162.820, Y  +613.309, Z    +0.000, E1   -63.489, E3 +225309.401}
SPL {X  -162.820, Y  +619.956, Z    +0.000, E1   -63.110, E3 +225319.088}
SPL {X  -162.820, Y  +631.846, Z    +0.000, E1   -63.529, E3 +225328.478}
SPL {X  -162.820, Y  +642.772, Z    +0.000, E1   -63.348, E3 +225341.281}
SPL {X  -162.820, Y  +658.642, Z    +0.000, E1   -63.324, E3 +225358.196}
SPL {X  -162.819, Y  +673.983, Z    +0.000, E1   -63.398, E3 +225373.524}
SPL {X  -162.399, Y  +685.202, Z    +0.000, E1   -63.235, E3 +225386.517}
SPL {X  -161.289, Y  +695.772, Z    +0.000, E1   -63.167, E3 +225397.967}
SPL {X  -160.212, Y  +702.527, Z    +0.000, E1   -62.898, E3 +225406.948}
SPL {X  -158.647, Y  +710.128, Z    +0.000, E1   -62.776, E3 +225415.771}
SPL {X  -156.957, Y  +716.799, Z    +0.000, E1   -62.460, E3 +225424.889}
SPL {X  -155.130, Y  +722.947, Z    +0.000, E1   -62.207, E3 +225433.001}
SPL {X  -152.287, Y  +731.112, Z    +0.000, E1   -61.798, E3 +225444.277}
SPL {X  -149.420, Y  +738.185, Z    +0.000, E1   -61.282, E3 +225454.685}
SPL {X  -146.033, Y  +745.504, Z    +0.000, E1   -60.844, E3 +225464.952}
SPL {X  -142.518, Y  +752.234, Z    +0.000, E1   -60.144, E3 +225475.579}
SPL {X  -138.778, Y  +758.653, Z    +0.000, E1   -59.483, E3 +225485.650}
SPL {X  -132.576, Y  +768.020, Z    +0.000, E1   -60.529, E3 +225490.411}
SPL {X  -102.851, Y  +799.722, Z    +0.000, E1   -53.923, E3 +225580.554}
SPL {X  -101.618, Y  +800.716, Z    +0.000, E1   -52.212, E3 +225693.539}
ENDSPLINE

SPLINE
SPL {X  -141.567, Y  +753.931, Z    +0.000, E1   -42.659, E3 +225730.242}
SPL {X  -155.442, Y  +721.958, Z    +0.000, E1   -30.769, E3 +225737.148}
SPL {X  -161.417, Y  +694.832, Z    +0.000, E1   -16.464, E3 +225741.117}
SPL {X  -162.719, Y  +679.228, Z    +0.000, E1    -6.085, E3 +225741.441}
SPL {X  -162.820, Y  +671.750, Z    +0.000, E1    -0.355, E3 +225740.878}
SPL {X  -162.820, Y  +669.853, Z    +0.000, E1    +1.938, E3 +225740.607}
SPL {X  -162.820, Y  +667.375, Z    +0.000, E1    +5.386, E3 +225740.444}
SPL {X  -162.820, Y  +663.189, Z    +0.000, E1   +11.952, E3 +225740.509}
SPL {X  -162.820, Y  +655.445, Z    +0.000, E1   +24.952, E3 +225740.455}
SPL {X  -162.820, Y  +644.088, Z    +0.000, E1   +41.840, E3 +225740.591}
SPL {X  -162.820, Y  +632.645, Z    +0.000, E1   +53.114, E3 +225741.327}
SPL {X  -162.820, Y  +584.142, Z    +0.000, E1   +66.966, E3 +225756.670}
SPL {X  -162.820, Y  +471.906, Z    +0.000, E1   +66.781, E3 +225838.911}
ENDSPLINE

SPLINE
SPL {X  -162.820, Y  +475.237, Z    +0.000, E1   +64.883, E3 +225850.598}
ENDSPLINE

SPLINE
SPL {X  -162.820, Y  +462.171, Z    +0.000, E1   +64.935, E3 +225863.084}
SPL {X  -162.820, Y  +448.581, Z    +0.000, E1   +64.948, E3 +225876.096}
SPL {X  -162.820, Y  +437.579, Z    +0.000, E1   +64.893, E3 +225887.272}
SPL {X  -162.820, Y  +425.248, Z    +0.000, E1   +64.950, E3 +225898.859}
SPL {X  -162.820, Y  +417.868, Z    +0.000, E1   +64.478, E3 +225909.678}
ENDSPLINE

SPLINE
SPL {X  -162.820, Y  +442.889, Z    +0.000, E1   +58.918, E3 +225921.858}
ENDSPLINE

SPLINE
SPL {X  -162.820, Y  +428.091, Z    +0.000, E1   +59.583, E3 +225935.630}
SPL {X  -162.820, Y  +410.436, Z    +0.000, E1   +60.611, E3 +225949.832}
SPL {X  -162.820, Y  +385.611, Z    +0.000, E1   +62.089, E3 +225967.729}
SPL {X  -162.597, Y  +371.985, Z    +0.000, E1   +62.420, E3 +225980.118}
SPL {X  -161.572, Y  +360.382, Z    +0.000, E1   +62.315, E3 +225993.689}
SPL {X  -160.005, Y  +350.357, Z    +0.000, E1   +62.043, E3 +226006.252}
SPL {X  -157.973, Y  +341.066, Z    +0.000, E1   +61.800, E3 +226018.169}
SPL {X  -155.627, Y  +332.640, Z    +0.000, E1   +61.354, E3 +226030.084}
SPL {X  -153.198, Y  +325.358, Z    +0.000, E1   +61.117, E3 +226039.514}
SPL {X  -151.022, Y  +319.651, Z    +0.000, E1   +60.776, E3 +226047.687}
SPL {X  -149.105, Y  +315.094, Z    +0.000, E1   +60.301, E3 +226055.440}
SPL {X  -146.196, Y  +308.826, Z    +0.000, E1   +59.961, E3 +226064.146}
SPL {X  -143.704, Y  +303.952, Z    +0.000, E1   +59.374, E3 +226072.503}
SPL {X  -140.940, Y  +298.976, Z    +0.000, E1   +59.075, E3 +226079.428}
SPL {X  -137.763, Y  +293.715, Z    +0.000, E1   +58.761, E3 +226086.535}
SPL {X  -129.725, Y  +282.103, Z    +0.000, E1   +61.069, E3 +226088.038}
SPL {X  -106.695, Y  +257.510, Z    +0.000, E1   +52.408, E3 +226188.761}
SPL {X  -104.122, Y  +255.325, Z    +0.000, E1   +51.312, E3 +226278.818}
ENDSPLINE

SPLINE
SPL {X  -140.007, Y  +297.383, Z    +0.000, E1   +42.766, E3 +226318.143}
SPL {X  -156.919, Y  +337.064, Z    +0.000, E1   +27.647, E3 +226324.294}
SPL {X  -160.736, Y  +354.534, Z    +0.000, E1   +18.553, E3 +226326.990}
SPL {X  -162.078, Y  +364.978, Z    +0.000, E1   +12.369, E3 +226328.675}
SPL {X  -162.656, Y  +373.196, Z    +0.000, E1    +6.960, E3 +226328.170}
SPL {X  -162.819, Y  +379.805, Z    +0.000, E1    +2.285, E3 +226328.294}
SPL {X  -162.820, Y  +383.416, Z    +0.000, E1    -0.722, E3 +226327.718}
SPL {X  -162.820, Y  +388.628, Z    +0.000, E1    -7.678, E3 +226327.486}
SPL {X  -162.820, Y  +394.643, Z    +0.000, E1   -17.317, E3 +226327.286}
SPL {X  -162.820, Y  +401.515, Z    +0.000, E1   -27.960, E3 +226328.107}
SPL {X  -162.820, Y  +412.105, Z    +0.000, E1   -42.847, E3 +226327.099}
SPL {X  -162.820, Y  +422.796, Z    +0.000, E1   -52.392, E3 +226328.319}
SPL {X  -162.820, Y  +474.423, Z    +0.000, E1   -65.078, E3 +226349.370}
SPL {X  -162.820, Y  +578.686, Z    +0.000, E1   -67.085, E3 +226418.535}
ENDSPLINE

SPLINE
SPL {X  -162.820, Y  +565.364, Z    +0.000, E1   -63.589, E3 +226432.535}
ENDSPLINE

SPLINE
SPL {X  -162.820, Y  +574.608, Z    +0.000, E1   -63.370, E3 +226443.793}
SPL {X  -162.820, Y  +584.314, Z    +0.000, E1   -63.342, E3 +226454.085}
SPL {X  -162.820, Y  +593.857, Z    +0.000, E1   -63.382, E3 +226463.788}
SPL {X  -162.820, Y  +602.272, Z    +0.000, E1   -63.279, E3 +226473.316}
SPL {X  -162.820, Y  +613.309, Z    +0.000, E1   -63.489, E3 +226483.314}
SPL {X  -162.820, Y  +619.956, Z    +0.000, E1   -63.110, E3 +226493.001}
SPL {X  -162.820, Y  +634.513, Z    +0.000, E1   -63.471, E3 +226505.767}
SPL {X  -162.820, Y  +648.936, Z    +0.000, E1   -63.278, E3 +226522.222}
SPL {X  -162.820, Y  +662.662, Z    +0.000, E1   -63.383, E3 +226535.714}
SPL {X  -162.819, Y  +673.983, Z    +0.000, E1   -63.398, E3 +226547.437}
SPL {X  -162.399, Y  +685.202, Z    +0.000, E1   -63.235, E3 +226560.431}
SPL {X  -161.289, Y  +695.772, Z    +0.000, E1   -63.167, E3 +226571.880}
SPL {X  -160.212, Y  +702.527, Z    +0.000, E1   -62.898, E3 +226580.861}
SPL {X  -158.647, Y  +710.128, Z    +0.000, E1   -62.776, E3 +226589.684}
SPL {X  -156.957, Y  +716.799, Z    +0.000, E1   -62.460, E3 +226598.802}
SPL {X  -154.447, Y  +725.041, Z    +0.000, E1   -62.170, E3 +226609.459}
SPL {X  -151.721, Y  +732.586, Z    +0.000, E1   -61.616, E3 +226620.709}
SPL {X  -149.420, Y  +738.185, Z    +0.000, E1   -61.282, E3 +226628.598}
SPL {X  -146.033, Y  +745.504, Z    +0.000, E1   -60.844, E3 +226638.865}
SPL {X  -142.518, Y  +752.234, Z    +0.000, E1   -60.144, E3 +226649.492}
SPL {X  -139.430, Y  +757.582, Z    +0.000, E1   -59.554, E3 +226658.023}
SPL {X  -135.510, Y  +763.762, Z    +0.000, E1   -59.735, E3 +226663.544}
SPL {X  -130.418, Y  +770.976, Z    +0.000, E1   -60.870, E3 +226665.701}
SPL {X  -100.103, Y  +801.912, Z    +0.000, E1   -53.794, E3 +226762.024}
ENDSPLINE

SPLINE
SPL {X  -112.938, Y  +790.784, Z    +0.000, E1   -51.983, E3 +226897.547}
SPL {X  -141.567, Y  +753.931, Z    +0.000, E1   -42.659, E3 +226904.155}
SPL {X  -155.442, Y  +721.958, Z    +0.000, E1   -30.769, E3 +226911.061}
SPL {X  -160.289, Y  +702.098, Z    +0.000, E1   -20.686, E3 +226914.789}
SPL {X  -162.312, Y  +686.349, Z    +0.000, E1   -11.031, E3 +226915.195}
SPL {X  -162.811, Y  +675.182, Z    +0.000, E1    -3.078, E3 +226915.269}
SPL {X  -162.820, Y  +671.474, Z    +0.000, E1    -0.022, E3 +226914.739}
SPL {X  -162.820, Y  +668.525, Z    +0.000, E1    +3.543, E3 +226914.433}
SPL {X  -162.820, Y  +663.189, Z    +0.000, E1   +11.952, E3 +226914.422}
SPL {X  -162.820, Y  +655.445, Z    +0.000, E1   +24.952, E3 +226914.368}
SPL {X  -162.820, Y  +644.088, Z    +0.000, E1   +41.840, E3 +226914.504}
SPL {X  -162.820, Y  +632.645, Z    +0.000, E1   +53.114, E3 +226915.240}
SPL {X  -162.820, Y  +584.142, Z    +0.000, E1   +66.966, E3 +226930.583}
SPL {X  -162.820, Y  +471.906, Z    +0.000, E1   +66.781, E3 +227012.824}
SPL {X  -162.820, Y  +470.218, Z    +0.000, E1   +64.979, E3 +227028.825}
SPL {X  -162.820, Y  +452.619, Z    +0.000, E1   +64.912, E3 +227046.503}
SPL {X  -162.820, Y  +437.579, Z    +0.000, E1   +64.893, E3 +227061.185}
SPL {X  -162.820, Y  +425.248, Z    +0.000, E1   +64.950, E3 +227072.772}
SPL {X  -162.820, Y  +417.868, Z    +0.000, E1   +64.478, E3 +227083.591}
ENDSPLINE

SPLINE
SPL {X  -162.820, Y  +447.149, Z    +0.000, E1   +58.721, E3 +227091.587}
ENDSPLINE

SPLINE
SPL {X  -162.820, Y  +431.862, Z    +0.000, E1   +59.419, E3 +227106.134}
SPL {X  -162.820, Y  +417.107, Z    +0.000, E1   +60.148, E3 +227118.945}
SPL {X  -162.820, Y  +398.797, Z    +0.000, E1   +61.348, E3 +227132.077}
SPL {X  -162.753, Y  +375.814, Z    +0.000, E1   +62.427, E3 +227149.999}
SPL {X  -161.572, Y  +360.382, Z    +0.000, E1   +62.315, E3 +227167.602}
SPL {X  -160.005, Y  +350.357, Z    +0.000, E1   +62.043, E3 +227180.165}
SPL {X  -158.606, Y  +343.697, Z    +0.000, E1   +61.897, E3 +227188.388}
SPL {X  -156.311, Y  +334.925, Z    +0.000, E1   +61.505, E3 +227200.735}
SPL {X  -153.198, Y  +325.358, Z    +0.000, E1   +61.117, E3 +227213.427}
SPL {X  -151.022, Y  +319.651, Z    +0.000, E1   +60.776, E3 +227221.600}
SPL {X  -149.105, Y  +315.094, Z    +0.000, E1   +60.301, E3 +227229.353}
SPL {X  -146.196, Y  +308.826, Z    +0.000, E1   +59.961, E3 +227238.059}
SPL {X  -143.704, Y  +303.952, Z    +0.000, E1   +59.374, E3 +227246.416}
SPL {X  -140.940, Y  +298.976, Z    +0.000, E1   +59.075, E3 +227253.342}
SPL {X  -137.763, Y  +293.715, Z    +0.000, E1   +58.761, E3 +227260.448}
SPL {X  -129.725, Y  +282.103, Z    +0.000, E1   +61.069, E3 +227261.951}
SPL {X  -106.695, Y  +257.510, Z    +0.000, E1   +52.408, E3 +227362.674}
SPL {X  -104.122, Y  +255.325, Z    +0.000, E1   +51.312, E3 +227452.732}
ENDSPLINE

SPLINE
SPL {X  -140.007, Y  +297.383, Z    +0.000, E1   +42.766, E3 +227492.056}
SPL {X  -155.551, Y  +332.393, Z    +0.000, E1   +29.794, E3 +227497.978}
SPL {X  -159.755, Y  +349.054, Z    +0.000, E1   +21.610, E3 +227499.851}
SPL {X  -162.078, Y  +364.978, Z    +0.000, E1   +12.369, E3 +227502.588}
SPL {X  -162.752, Y  +375.778, Z    +0.000, E1    +5.236, E3 +227502.297}
SPL {X  -162.820, Y  +381.939, Z    +0.000, E1    +0.593, E3 +227501.924}
SPL {X  -162.820, Y  +383.993, Z    +0.000, E1    -1.497, E3 +227501.497}
SPL {X  -162.820, Y  +388.628, Z    +0.000, E1    -7.678, E3 +227501.399}
SPL {X  -162.820, Y  +394.643, Z    +0.000, E1   -17.317, E3 +227501.199}
SPL {X  -162.820, Y  +401.515, Z    +0.000, E1   -27.960, E3 +227502.020}
SPL {X  -162.820, Y  +412.105, Z    +0.000, E1   -42.847, E3 +227501.012}
SPL {X  -162.820, Y  +422.796, Z    +0.000, E1   -52.392, E3 +227502.232}
SPL {X  -162.820, Y  +474.423, Z    +0.000, E1   -65.078, E3 +227523.283}
SPL {X  -162.820, Y  +578.686, Z    +0.000, E1   -67.085, E3 +227592.448}
ENDSPLINE

SPLINE
SPL {X  -162.820, Y  +565.364, Z    +0.000, E1   -63.589, E3 +227606.448}
ENDSPLINE

SPLINE
SPL {X  -162.820, Y  +574.608, Z    +0.000, E1   -63.370, E3 +227617.706}
SPL {X  -162.820, Y  +584.314, Z    +0.000, E1   -63.342, E3 +227627.998}
SPL {X  -162.820, Y  +593.857, Z    +0.000, E1   -63.382, E3 +227637.701}
SPL {X  -162.820, Y  +602.272, Z    +0.000, E1   -63.279, E3 +227647.229}
SPL {X  -162.820, Y  +613.309, Z    +0.000, E1   -63.489, E3 +227657.228}
SPL {X  -162.820, Y  +627.013, Z    +0.000, E1   -63.389, E3 +227672.449}
SPL {X  -162.820, Y  +642.772, Z    +0.000, E1   -63.348, E3 +227689.107}
SPL {X  -162.820, Y  +658.642, Z    +0.000, E1   -63.324, E3 +227706.022}
SPL {X  -162.819, Y  +673.983, Z    +0.000, E1   -63.398, E3 +227721.350}
SPL {X  -162.617, Y  +681.634, Z    +0.000, E1   -63.169, E3 +227730.972}
SPL {X  -161.618, Y  +693.246, Z    +0.000, E1   -63.233, E3 +227742.829}
SPL {X  -160.212, Y  +702.527, Z    +0.000, E1   -62.898, E3 +227754.774}
SPL {X  -158.647, Y  +710.128, Z    +0.000, E1   -62.776, E3 +227763.597}
SPL {X  -156.957, Y  +716.799, Z    +0.000, E1   -62.460, E3 +227772.715}
SPL {X  -155.130, Y  +722.947, Z    +0.000, E1   -62.207, E3 +227780.827}
SPL {X  -152.287, Y  +731.112, Z    +0.000, E1   -61.798, E3 +227792.103}
SPL {X  -149.420, Y  +738.185, Z    +0.000, E1   -61.282, E3 +227802.511}
SPL {X  -146.033, Y  +745.504, Z    +0.000, E1   -60.844, E3 +227812.778}
SPL {X  -142.518, Y  +752.234, Z    +0.000, E1   -60.144, E3 +227823.405}
SPL {X  -139.430, Y  +757.582, Z    +0.000, E1   -59.554, E3 +227831.937}
SPL {X  -134.550, Y  +765.187, Z    +0.000, E1   -59.954, E3 +227837.888}
SPL {X  -100.103, Y  +801.912, Z    +0.000, E1   -53.794, E3 +227935.937}
ENDSPLINE

SPLINE
SPL {X  -112.938, Y  +790.784, Z    +0.000, E1   -51.983, E3 +228071.460}
SPL {X  -141.567, Y  +753.931, Z    +0.000, E1   -42.659, E3 +228078.068}
SPL {X  -155.442, Y  +721.958, Z    +0.000, E1   -30.769, E3 +228084.974}
SPL {X  -161.417, Y  +694.832, Z    +0.000, E1   -16.464, E3 +228088.943}
SPL {X  -162.719, Y  +679.228, Z    +0.000, E1    -6.085, E3 +228089.267}
SPL {X  -162.820, Y  +673.638, Z    +0.000, E1    -1.806, E3 +228089.057}
SPL {X  -162.820, Y  +670.948, Z    +0.000, E1    +0.412, E3 +228088.581}
SPL {X  -162.820, Y  +667.375, Z    +0.000, E1    +5.386, E3 +228088.270}
SPL {X  -162.820, Y  +663.189, Z    +0.000, E1   +11.952, E3 +228088.335}
SPL {X  -162.820, Y  +655.445, Z    +0.000, E1   +24.952, E3 +228088.281}
SPL {X  -162.820, Y  +644.088, Z    +0.000, E1   +41.840, E3 +228088.417}
SPL {X  -162.820, Y  +632.645, Z    +0.000, E1   +53.114, E3 +228089.153}
SPL {X  -162.820, Y  +584.142, Z    +0.000, E1   +66.966, E3 +228104.496}
SPL {X  -162.820, Y  +466.182, Z    +0.000, E1   +68.456, E3 +228178.266}
ENDSPLINE

SPLINE
SPL {X  -162.820, Y  +475.083, Z    +0.000, E1   +65.244, E3 +228195.967}
ENDSPLINE

SPLINE
SPL {X  -162.820, Y  +465.389, Z    +0.000, E1   +65.015, E3 +228206.984}
SPL {X  -162.820, Y  +452.619, Z    +0.000, E1   +64.912, E3 +228220.416}
SPL {X  -162.820, Y  +437.579, Z    +0.000, E1   +64.893, E3 +228235.098}
SPL {X  -162.820, Y  +425.248, Z    +0.000, E1   +64.950, E3 +228246.685}
SPL {X  -162.820, Y  +417.868, Z    +0.000, E1   +64.478, E3 +228257.504}
ENDSPLINE

SPLINE
SPL {X  -162.820, Y  +442.889, Z    +0.000, E1   +58.918, E3 +228269.684}
ENDSPLINE

SPLINE
SPL {X  -162.820, Y  +428.091, Z    +0.000, E1   +59.583, E3 +228283.456}
SPL {X  -162.820, Y  +417.107, Z    +0.000, E1   +60.148, E3 +228292.858}
SPL {X  -162.820, Y  +398.797, Z    +0.000, E1   +61.348, E3 +228305.990}
SPL {X  -162.819, Y  +379.881, Z    +0.000, E1   +62.356, E3 +228319.820}
SPL {X  -162.597, Y  +371.985, Z    +0.000, E1   +62.420, E3 +228327.944}
SPL {X  -161.953, Y  +363.716, Z    +0.000, E1   +62.355, E3 +228337.401}
SPL {X  -160.528, Y  +353.277, Z    +0.000, E1   +62.144, E3 +228350.397}
SPL {X  -158.606, Y  +343.697, Z    +0.000, E1   +61.897, E3 +228362.301}
SPL {X  -156.311, Y  +334.925, Z    +0.000, E1   +61.505, E3 +228374.648}
SPL {X  -153.198, Y  +325.358, Z    +0.000, E1   +61.117, E3 +228387.340}
SPL {X  -151.022, Y  +319.651, Z    +0.000, E1   +60.776, E3 +228395.513}
SPL {X  -149.105, Y  +315.094, Z    +0.000, E1   +60.301, E3 +228403.266}
SPL {X  -146.196, Y  +308.826, Z    +0.000, E1   +59.961, E3 +228411.972}
SPL {X  -143.704, Y  +303.952, Z    +0.000, E1   +59.374, E3 +228420.330}
SPL {X  -140.940, Y  +298.976, Z    +0.000, E1   +59.075, E3 +228427.255}
SPL {X  -137.763, Y  +293.715, Z    +0.000, E1   +58.761, E3 +228434.361}
SPL {X  -129.725, Y  +282.103, Z    +0.000, E1   +61.069, E3 +228435.864}
SPL {X  -106.695, Y  +257.510, Z    +0.000, E1   +52.408, E3 +228536.587}
SPL {X  -104.122, Y  +255.325, Z    +0.000, E1   +51.312, E3 +228626.645}
ENDSPLINE

SPLINE
SPL {X  -140.007, Y  +297.383, Z    +0.000, E1   +42.766, E3 +228665.969}
SPL {X  -156.919, Y  +337.064, Z    +0.000, E1   +27.647, E3 +228672.120}
SPL {X  -160.736, Y  +354.534, Z    +0.000, E1   +18.553, E3 +228674.816}
SPL {X  -162.078, Y  +364.978, Z    +0.000, E1   +12.369, E3 +228676.501}
SPL {X  -162.656, Y  +373.196, Z    +0.000, E1    +6.960, E3 +228675.996}
SPL {X  -162.819, Y  +379.805, Z    +0.000, E1    +2.285, E3 +228676.120}
SPL {X  -162.820, Y  +382.398, Z    +0.000, E1    +0.126, E3 +228675.780}
SPL {X  -162.820, Y  +383.993, Z    +0.000, E1    -1.497, E3 +228675.410}
SPL {X  -162.820, Y  +387.367, Z    +0.000, E1    -6.003, E3 +228675.416}
SPL {X  -162.820, Y  +390.506, Z    +0.000, E1   -10.770, E3 +228675.159}
SPL {X  -162.820, Y  +394.643, Z    +0.000, E1   -17.317, E3 +228675.112}
SPL {X  -162.820, Y  +401.515, Z    +0.000, E1   -27.960, E3 +228675.933}
SPL {X  -162.820, Y  +412.105, Z    +0.000, E1   -42.847, E3 +228674.925}
SPL {X  -162.820, Y  +422.796, Z    +0.000, E1   -52.392, E3 +228676.145}
SPL {X  -162.820, Y  +474.423, Z    +0.000, E1   -65.078, E3 +228697.196}
SPL {X  -162.820, Y  +578.686, Z    +0.000, E1   -67.085, E3 +228766.361}
ENDSPLINE

SPLINE
SPL {X  -162.820, Y  +565.364, Z    +0.000, E1   -63.589, E3 +228780.361}
ENDSPLINE

SPLINE
SPL {X  -162.820, Y  +574.608, Z    +0.000, E1   -63.370, E3 +228791.619}
SPL {X  -162.820, Y  +584.314, Z    +0.000, E1   -63.342, E3 +228801.911}
SPL {X  -162.820, Y  +593.857, Z    +0.000, E1   -63.382, E3 +228811.614}
SPL {X  -162.820, Y  +602.272, Z    +0.000, E1   -63.279, E3 +228821.142}
SPL {X  -162.820, Y  +613.309, Z    +0.000, E1   -63.489, E3 +228831.141}
SPL {X  -162.820, Y  +619.956, Z    +0.000, E1   -63.110, E3 +228840.827}
SPL {X  -162.820, Y  +634.513, Z    +0.000, E1   -63.471, E3 +228853.593}
SPL {X  -162.820, Y  +648.936, Z    +0.000, E1   -63.278, E3 +228870.048}
SPL {X  -162.820, Y  +662.662, Z    +0.000, E1   -63.383, E3 +228883.540}
SPL {X  -162.819, Y  +673.983, Z    +0.000, E1   -63.398, E3 +228895.263}
SPL {X  -162.617, Y  +681.634, Z    +0.000, E1   -63.169, E3 +228904.885}
SPL {X  -161.618, Y  +693.246, Z    +0.000, E1   -63.233, E3 +228916.742}
SPL {X  -160.212, Y  +702.527, Z    +0.000, E1   -62.898, E3 +228928.687}
SPL {X  -158.647, Y  +710.128, Z    +0.000, E1   -62.776, E3 +228937.510}
SPL {X  -156.957, Y  +716.799, Z    +0.000, E1   -62.460, E3 +228946.628}
SPL {X  -154.447, Y  +725.041, Z    +0.000, E1   -62.170, E3 +228957.285}
SPL {X  -151.721, Y  +732.586, Z    +0.000, E1   -61.616, E3 +228968.535}
SPL {X  -149.420, Y  +738.185, Z    +0.000, E1   -61.282, E3 +228976.424}
SPL {X  -146.033, Y  +745.504, Z    +0.000, E1   -60.844, E3 +228986.691}
SPL {X  -142.518, Y  +752.234, Z    +0.000, E1   -60.144, E3 +228997.318}
SPL {X  -138.778, Y  +758.653, Z    +0.000, E1   -59.483, E3 +229007.389}
SPL {X  -132.576, Y  +768.020, Z    +0.000, E1   -60.529, E3 +229012.151}
SPL {X  -100.103, Y  +801.912, Z    +0.000, E1   -53.794, E3 +229109.850}
ENDSPLINE

SPLINE
SPL {X  -112.938, Y  +790.784, Z    +0.000, E1   -51.983, E3 +229245.373}
SPL {X  -145.058, Y  +747.450, Z    +0.000, E1   -40.634, E3 +229253.483}
SPL {X  -158.857, Y  +709.206, Z    +0.000, E1   -24.633, E3 +229261.452}
SPL {X  -162.312, Y  +686.349, Z    +0.000, E1   -11.031, E3 +229263.021}
SPL {X  -162.811, Y  +675.182, Z    +0.000, E1    -3.078, E3 +229263.095}
SPL {X  -162.820, Y  +671.474, Z    +0.000, E1    -0.022, E3 +229262.565}
SPL {X  -162.820, Y  +668.525, Z    +0.000, E1    +3.543, E3 +229262.259}
SPL {X  -162.820, Y  +663.189, Z    +0.000, E1   +11.952, E3 +229262.248}
SPL {X  -162.820, Y  +657.986, Z    +0.000, E1   +20.997, E3 +229261.962}
SPL {X  -162.820, Y  +650.033, Z    +0.000, E1   +33.465, E3 +229262.431}
SPL {X  -162.820, Y  +635.632, Z    +0.000, E1   +50.654, E3 +229262.756}
SPL {X  -162.820, Y  +584.142, Z    +0.000, E1   +66.966, E3 +229278.409}
SPL {X  -162.820, Y  +471.906, Z    +0.000, E1   +66.781, E3 +229360.650}
SPL {X  -162.820, Y  +470.218, Z    +0.000, E1   +64.979, E3 +229376.651}
SPL {X  -162.820, Y  +452.619, Z    +0.000, E1   +64.912, E3 +229394.329}
SPL {X  -162.820, Y  +437.579, Z    +0.000, E1   +64.893, E3 +229409.011}
SPL {X  -162.820, Y  +425.248, Z    +0.000, E1   +64.950, E3 +229420.598}
SPL {X  -162.820, Y  +417.868, Z    +0.000, E1   +64.478, E3 +229431.417}
ENDSPLINE

SPLINE
SPL {X  -162.820, Y  +447.149, Z    +0.000, E1   +58.721, E3 +229439.413}
ENDSPLINE

SPLINE
SPL {X  -162.820, Y  +431.862, Z    +0.000, E1   +59.419, E3 +229453.960}
SPL {X  -162.820, Y  +417.107, Z    +0.000, E1   +60.148, E3 +229466.771}
SPL {X  -162.820, Y  +398.797, Z    +0.000, E1   +61.348, E3 +229479.903}
SPL {X  -162.753, Y  +375.814, Z    +0.000, E1   +62.427, E3 +229497.825}
SPL {X  -161.572, Y  +360.382, Z    +0.000, E1   +62.315, E3 +229515.428}
SPL {X  -160.005, Y  +350.357, Z    +0.000, E1   +62.043, E3 +229527.991}
SPL {X  -158.606, Y  +343.697, Z    +0.000, E1   +61.897, E3 +229536.214}
SPL {X  -156.311, Y  +334.925, Z    +0.000, E1   +61.505, E3 +229548.561}
SPL {X  -153.198, Y  +325.358, Z    +0.000, E1   +61.117, E3 +229561.253}
SPL {X  -151.022, Y  +319.651, Z    +0.000, E1   +60.776, E3 +229569.426}
SPL {X  -149.105, Y  +315.094, Z    +0.000, E1   +60.301, E3 +229577.179}
SPL {X  -146.196, Y  +308.826, Z    +0.000, E1   +59.961, E3 +229585.885}
SPL {X  -143.704, Y  +303.952, Z    +0.000, E1   +59.374, E3 +229594.243}
SPL {X  -140.940, Y  +298.976, Z    +0.000, E1   +59.075, E3 +229601.168}
SPL {X  -137.763, Y  +293.715, Z    +0.000, E1   +58.761, E3 +229608.274}
SPL {X  -129.725, Y  +282.103, Z    +0.000, E1   +61.069, E3 +229609.777}
SPL {X  -106.695, Y  +257.510, Z    +0.000, E1   +52.408, E3 +229710.500}
SPL {X  -104.122, Y  +255.325, Z    +0.000, E1   +51.312, E3 +229800.558}
ENDSPLINE

SPLINE
SPL {X  -140.007, Y  +297.383, Z    +0.000, E1   +42.766, E3 +229839.882}
SPL {X  -155.551, Y  +332.393, Z    +0.000, E1   +29.794, E3 +229845.804}
SPL {X  -159.755, Y  +349.054, Z    +0.000, E1   +21.610, E3 +229847.677}
SPL {X  -162.078, Y  +364.978, Z    +0.000, E1   +12.369, E3 +229850.414}
SPL {X  -162.752, Y  +375.778, Z    +0.000, E1    +5.236, E3 +229850.123}
SPL {X  -162.820, Y  +381.939, Z    +0.000, E1    +0.593, E3 +229849.750}
SPL {X  -162.820, Y  +383.993, Z    +0.000, E1    -1.497, E3 +229849.323}
SPL {X  -162.820, Y  +388.628, Z    +0.000, E1    -7.678, E3 +229849.226}
SPL {X  -162.820, Y  +394.643, Z    +0.000, E1   -17.317, E3 +229849.025}
SPL {X  -162.820, Y  +401.515, Z    +0.000, E1   -27.960, E3 +229849.846}
SPL {X  -162.820, Y  +412.105, Z    +0.000, E1   -42.847, E3 +229848.838}
SPL {X  -162.820, Y  +422.796, Z    +0.000, E1   -52.392, E3 +229850.058}
SPL {X  -162.820, Y  +474.423, Z    +0.000, E1   -65.078, E3 +229871.109}
SPL {X  -162.820, Y  +578.686, Z    +0.000, E1   -67.085, E3 +229940.274}
ENDSPLINE

SPLINE
SPL {X  -162.820, Y  +565.364, Z    +0.000, E1   -63.589, E3 +229954.274}
ENDSPLINE

SPLINE
SPL {X  -162.820, Y  +574.608, Z    +0.000, E1   -63.370, E3 +229965.532}
SPL {X  -162.820, Y  +584.314, Z    +0.000, E1   -63.342, E3 +229975.824}
SPL {X  -162.820, Y  +593.857, Z    +0.000, E1   -63.382, E3 +229985.527}
SPL {X  -162.820, Y  +602.272, Z    +0.000, E1   -63.279, E3 +229995.055}
SPL {X  -162.820, Y  +613.309, Z    +0.000, E1   -63.489, E3 +230005.054}
SPL {X  -162.820, Y  +627.013, Z    +0.000, E1   -63.389, E3 +230020.275}
SPL {X  -162.820, Y  +642.772, Z    +0.000, E1   -63.348, E3 +230036.933}
SPL {X  -162.820, Y  +658.642, Z    +0.000, E1   -63.324, E3 +230053.848}
SPL {X  -162.819, Y  +673.983, Z    +0.000, E1   -63.398, E3 +230069.176}
SPL {X  -162.617, Y  +681.634, Z    +0.000, E1   -63.169, E3 +230078.798}
SPL {X  -161.618, Y  +693.246, Z    +0.000, E1   -63.233, E3 +230090.655}
SPL {X  -160.212, Y  +702.527, Z    +0.000, E1   -62.898, E3 +230102.600}
SPL {X  -158.647, Y  +710.128, Z    +0.000, E1   -62.776, E3 +230111.423}
SPL {X  -156.957, Y  +716.799, Z    +0.000, E1   -62.460, E3 +230120.541}
SPL {X  -155.130, Y  +722.947, Z    +0.000, E1   -62.207, E3 +230128.653}
SPL {X  -152.287, Y  +731.112, Z    +0.000, E1   -61.798, E3 +230139.929}
SPL {X  -149.420, Y  +738.185, Z    +0.000, E1   -61.282, E3 +230150.337}
SPL {X  -146.960, Y  +743.593, Z    +0.000, E1   -60.951, E3 +230157.881}
SPL {X  -143.277, Y  +750.844, Z    +0.000, E1   -60.348, E3 +230168.888}
SPL {X  -139.430, Y  +757.582, Z    +0.000, E1   -59.554, E3 +230179.763}
SPL {X  -134.550, Y  +765.187, Z    +0.000, E1   -59.954, E3 +230185.714}
SPL {X  -100.103, Y  +801.912, Z    +0.000, E1   -53.794, E3 +230283.764}
ENDSPLINE

SPLINE
SPL {X  -112.938, Y  +790.784, Z    +0.000, E1   -51.983, E3 +230419.286}
SPL {X  -145.058, Y  +747.450, Z    +0.000, E1   -40.634, E3 +230427.396}
SPL {X  -158.857, Y  +709.206, Z    +0.000, E1   -24.633, E3 +230435.365}
SPL {X  -162.312, Y  +686.349, Z    +0.000, E1   -11.031, E3 +230436.934}
SPL {X  -162.811, Y  +675.182, Z    +0.000, E1    -3.078, E3 +230437.008}
SPL {X  -162.820, Y  +671.474, Z    +0.000, E1    -0.022, E3 +230436.478}
SPL {X  -162.820, Y  +668.525, Z    +0.000, E1    +3.543, E3 +230436.172}
SPL {X  -162.820, Y  +663.189, Z    +0.000, E1   +11.952, E3 +230436.161}
SPL {X  -162.820, Y  +657.986, Z    +0.000, E1   +20.997, E3 +230435.875}
SPL {X  -162.820, Y  +650.033, Z    +0.000, E1   +33.465, E3 +230436.344}
SPL {X  -162.820, Y  +635.632, Z    +0.000, E1   +50.654, E3 +230436.669}
SPL {X  -162.820, Y  +584.142, Z    +0.000, E1   +66.966, E3 +230452.322}
SPL {X  -162.820, Y  +471.906, Z    +0.000, E1   +66.781, E3 +230534.563}
SPL {X  -162.820, Y  +470.218, Z    +0.000, E1   +64.979, E3 +230550.564}
SPL {X  -162.820, Y  +452.619, Z    +0.000, E1   +64.912, E3 +230568.242}
SPL {X  -162.820, Y  +437.579, Z    +0.000, E1   +64.893, E3 +230582.924}
SPL {X  -162.820, Y  +425.248, Z    +0.000, E1   +64.950, E3 +230594.511}
SPL {X  -162.820, Y  +417.868, Z    +0.000, E1   +64.478, E3 +230605.330}
ENDSPLINE

SPLINE
SPL {X  -162.820, Y  +447.149, Z    +0.000, E1   +58.721, E3 +230613.326}
ENDSPLINE

SPLINE
SPL {X  -162.820, Y  +431.862, Z    +0.000, E1   +59.419, E3 +230627.873}
SPL {X  -162.820, Y  +417.107, Z    +0.000, E1   +60.148, E3 +230640.684}
SPL {X  -162.820, Y  +398.797, Z    +0.000, E1   +61.348, E3 +230653.816}
SPL {X  -162.753, Y  +375.814, Z    +0.000, E1   +62.427, E3 +230671.738}
SPL {X  -161.572, Y  +360.382, Z    +0.000, E1   +62.315, E3 +230689.341}
SPL {X  -160.005, Y  +350.357, Z    +0.000, E1   +62.043, E3 +230701.904}
SPL {X  -158.606, Y  +343.697, Z    +0.000, E1   +61.897, E3 +230710.127}
SPL {X  -156.311, Y  +334.925, Z    +0.000, E1   +61.505, E3 +230722.474}
SPL {X  -153.198, Y  +325.358, Z    +0.000, E1   +61.117, E3 +230735.166}
SPL {X  -151.022, Y  +319.651, Z    +0.000, E1   +60.776, E3 +230743.339}
SPL {X  -149.105, Y  +315.094, Z    +0.000, E1   +60.301, E3 +230751.092}
SPL {X  -146.196, Y  +308.826, Z    +0.000, E1   +59.961, E3 +230759.798}
SPL {X  -143.704, Y  +303.952, Z    +0.000, E1   +59.374, E3 +230768.156}
SPL {X  -140.940, Y  +298.976, Z    +0.000, E1   +59.075, E3 +230775.081}
SPL {X  -137.763, Y  +293.715, Z    +0.000, E1   +58.761, E3 +230782.187}
SPL {X  -129.725, Y  +282.103, Z    +0.000, E1   +61.069, E3 +230783.690}
SPL {X  -106.695, Y  +257.510, Z    +0.000, E1   +52.408, E3 +230884.413}
SPL {X  -104.122, Y  +255.325, Z    +0.000, E1   +51.312, E3 +230974.471}
ENDSPLINE

SPLINE
SPL {X  -140.007, Y  +297.383, Z    +0.000, E1   +42.766, E3 +231013.795}
SPL {X  -155.551, Y  +332.393, Z    +0.000, E1   +29.794, E3 +231019.717}
SPL {X  -159.755, Y  +349.054, Z    +0.000, E1   +21.610, E3 +231021.590}
SPL {X  -162.078, Y  +364.978, Z    +0.000, E1   +12.369, E3 +231024.327}
SPL {X  -162.752, Y  +375.778, Z    +0.000, E1    +5.236, E3 +231024.036}
SPL {X  -162.820, Y  +381.939, Z    +0.000, E1    +0.593, E3 +231023.663}
SPL {X  -162.820, Y  +383.993, Z    +0.000, E1    -1.497, E3 +231023.236}
SPL {X  -162.820, Y  +388.628, Z    +0.000, E1    -7.678, E3 +231023.139}
SPL {X  -162.820, Y  +394.643, Z    +0.000, E1   -17.317, E3 +231022.938}
SPL {X  -162.820, Y  +401.515, Z    +0.000, E1   -27.960, E3 +231023.759}
SPL {X  -162.820, Y  +412.105, Z    +0.000, E1   -42.847, E3 +231022.751}
SPL {X  -162.820, Y  +422.796, Z    +0.000, E1   -52.392, E3 +231023.971}
SPL {X  -162.820, Y  +474.423, Z    +0.000, E1   -65.078, E3 +231045.022}
SPL {X  -162.820, Y  +578.686, Z    +0.000, E1   -67.085, E3 +231114.187}
ENDSPLINE

SPLINE
SPL {X  -162.820, Y  +565.364, Z    +0.000, E1   -63.589, E3 +231128.187}
ENDSPLINE

SPLINE
SPL {X  -162.820, Y  +574.608, Z    +0.000, E1   -63.370, E3 +231139.445}
SPL {X  -162.820, Y  +584.314, Z    +0.000, E1   -63.342, E3 +231149.737}
SPL {X  -162.820, Y  +593.857, Z    +0.000, E1   -63.382, E3 +231159.440}
SPL {X  -162.820, Y  +602.272, Z    +0.000, E1   -63.279, E3 +231168.968}
SPL {X  -162.820, Y  +613.309, Z    +0.000, E1   -63.489, E3 +231178.967}
SPL {X  -162.820, Y  +619.956, Z    +0.000, E1   -63.110, E3 +231188.653}
SPL {X  -162.820, Y  +631.846, Z    +0.000, E1   -63.529, E3 +231198.044}
SPL {X  -162.820, Y  +642.772, Z    +0.000, E1   -63.348, E3 +231210.846}
SPL {X  -162.820, Y  +658.642, Z    +0.000, E1   -63.324, E3 +231227.761}
SPL {X  -162.819, Y  +673.983, Z    +0.000, E1   -63.398, E3 +231243.089}
SPL {X  -162.399, Y  +685.202, Z    +0.000, E1   -63.235, E3 +231256.083}
SPL {X  -161.289, Y  +695.772, Z    +0.000, E1   -63.167, E3 +231267.532}
SPL {X  -160.212, Y  +702.527, Z    +0.000, E1   -62.898, E3 +231276.513}
SPL {X  -158.647, Y  +710.128, Z    +0.000, E1   -62.776, E3 +231285.336}
SPL {X  -156.957, Y  +716.799, Z    +0.000, E1   -62.460, E3 +231294.454}
SPL {X  -154.447, Y  +725.041, Z    +0.000, E1   -62.170, E3 +231305.111}
SPL {X  -151.721, Y  +732.586, Z    +0.000, E1   -61.616, E3 +231316.361}
SPL {X  -149.420, Y  +738.185, Z    +0.000, E1   -61.282, E3 +231324.250}
SPL {X  -146.960, Y  +743.593, Z    +0.000, E1   -60.951, E3 +231331.794}
SPL {X  -143.277, Y  +750.844, Z    +0.000, E1   -60.348, E3 +231342.801}
SPL {X  -139.430, Y  +757.582, Z    +0.000, E1   -59.554, E3 +231353.676}
SPL {X  -134.550, Y  +765.187, Z    +0.000, E1   -59.954, E3 +231359.627}
SPL {X  -100.103, Y  +801.912, Z    +0.000, E1   -53.794, E3 +231457.677}
ENDSPLINE

SPLINE
SPL {X  -112.938, Y  +790.784, Z    +0.000, E1   -51.983, E3 +231593.199}
SPL {X  -141.567, Y  +753.931, Z    +0.000, E1   -42.659, E3 +231599.807}
SPL {X  -155.442, Y  +721.958, Z    +0.000, E1   -30.769, E3 +231606.713}
SPL {X  -161.417, Y  +694.832, Z    +0.000, E1   -16.464, E3 +231610.682}
SPL {X  -162.719, Y  +679.228, Z    +0.000, E1    -6.085, E3 +231611.006}
SPL {X  -162.820, Y  +673.638, Z    +0.000, E1    -1.806, E3 +231610.796}
SPL {X  -162.820, Y  +670.948, Z    +0.000, E1    +0.412, E3 +231610.320}
SPL {X  -162.820, Y  +667.375, Z    +0.000, E1    +5.386, E3 +231610.010}
SPL {X  -162.820, Y  +663.189, Z    +0.000, E1   +11.952, E3 +231610.074}
SPL {X  -162.820, Y  +655.445, Z    +0.000, E1   +24.952, E3 +231610.020}
SPL {X  -162.820, Y  +644.088, Z    +0.000, E1   +41.840, E3 +231610.157}
SPL {X  -162.820, Y  +632.645, Z    +0.000, E1   +53.114, E3 +231610.892}
SPL {X  -162.820, Y  +584.142, Z    +0.000, E1   +66.966, E3 +231626.235}
SPL {X  -162.820, Y  +471.906, Z    +0.000, E1   +66.781, E3 +231708.476}
SPL {X  -162.820, Y  +470.218, Z    +0.000, E1   +64.979, E3 +231724.477}
SPL {X  -162.820, Y  +452.619, Z    +0.000, E1   +64.912, E3 +231742.155}
SPL {X  -162.820, Y  +437.579, Z    +0.000, E1   +64.893, E3 +231756.837}
SPL {X  -162.820, Y  +425.248, Z    +0.000, E1   +64.950, E3 +231768.424}
SPL {X  -162.820, Y  +417.868, Z    +0.000, E1   +64.478, E3 +231779.243}
ENDSPLINE

SPLINE
SPL {X  -162.820, Y  +447.149, Z    +0.000, E1   +58.721, E3 +231787.239}
ENDSPLINE

SPLINE
SPL {X  -162.820, Y  +431.862, Z    +0.000, E1   +59.419, E3 +231801.786}
SPL {X  -162.820, Y  +417.107, Z    +0.000, E1   +60.148, E3 +231814.597}
SPL {X  -162.820, Y  +398.797, Z    +0.000, E1   +61.348, E3 +231827.729}
SPL {X  -162.753, Y  +375.814, Z    +0.000, E1   +62.427, E3 +231845.651}
SPL {X  -161.953, Y  +363.716, Z    +0.000, E1   +62.355, E3 +231859.140}
SPL {X  -160.528, Y  +353.277, Z    +0.000, E1   +62.144, E3 +231872.136}
SPL {X  -157.973, Y  +341.066, Z    +0.000, E1   +61.800, E3 +231887.735}
SPL {X  -155.627, Y  +332.640, Z    +0.000, E1   +61.354, E3 +231899.649}
SPL {X  -153.198, Y  +325.358, Z    +0.000, E1   +61.117, E3 +231909.079}
SPL {X  -151.022, Y  +319.651, Z    +0.000, E1   +60.776, E3 +231917.252}
SPL {X  -149.105, Y  +315.094, Z    +0.000, E1   +60.301, E3 +231925.005}
SPL {X  -146.196, Y  +308.826, Z    +0.000, E1   +59.961, E3 +231933.711}
SPL {X  -143.704, Y  +303.952, Z    +0.000, E1   +59.374, E3 +231942.069}
SPL {X  -140.940, Y  +298.976, Z    +0.000, E1   +59.075, E3 +231948.994}
SPL {X  -137.763, Y  +293.715, Z    +0.000, E1   +58.761, E3 +231956.100}
SPL {X  -129.725, Y  +282.103, Z    +0.000, E1   +61.069, E3 +231957.604}
SPL {X  -106.695, Y  +257.510, Z    +0.000, E1   +52.408, E3 +232058.326}
SPL {X  -104.122, Y  +255.325, Z    +0.000, E1   +51.312, E3 +232148.384}
ENDSPLINE

SPLINE
SPL {X  -140.007, Y  +297.383, Z    +0.000, E1   +42.766, E3 +232187.708}
SPL {X  -156.919, Y  +337.064, Z    +0.000, E1   +27.647, E3 +232193.859}
SPL {X  -161.737, Y  +361.753, Z    +0.000, E1   +14.421, E3 +232197.757}
SPL {X  -162.752, Y  +375.778, Z    +0.000, E1    +5.236, E3 +232197.949}
SPL {X  -162.820, Y  +382.443, Z    +0.000, E1    +0.212, E3 +232197.429}
SPL {X  -162.820, Y  +386.214, Z    +0.000, E1    -4.241, E3 +232197.131}
SPL {X  -162.820, Y  +390.506, Z    +0.000, E1   -10.770, E3 +232196.898}
SPL {X  -162.820, Y  +394.643, Z    +0.000, E1   -17.317, E3 +232196.852}
SPL {X  -162.820, Y  +401.515, Z    +0.000, E1   -27.960, E3 +232197.672}
SPL {X  -162.820, Y  +412.105, Z    +0.000, E1   -42.847, E3 +232196.664}
SPL {X  -162.820, Y  +422.796, Z    +0.000, E1   -52.392, E3 +232197.884}
SPL {X  -162.820, Y  +474.423, Z    +0.000, E1   -65.078, E3 +232218.935}
SPL {X  -162.820, Y  +578.686, Z    +0.000, E1   -67.085, E3 +232288.100}
ENDSPLINE

SPLINE
SPL {X  -162.820, Y  +565.364, Z    +0.000, E1   -63.589, E3 +232302.100}
ENDSPLINE

SPLINE
SPL {X  -162.820, Y  +574.608, Z    +0.000, E1   -63.370, E3 +232313.359}
SPL {X  -162.820, Y  +584.314, Z    +0.000, E1   -63.342, E3 +232323.651}
SPL {X  -162.820, Y  +593.857, Z    +0.000, E1   -63.382, E3 +232333.353}
SPL {X  -162.820, Y  +602.272, Z    +0.000, E1   -63.279, E3 +232342.881}
SPL {X  -162.820, Y  +613.309, Z    +0.000, E1   -63.489, E3 +232352.880}
SPL {X  -162.820, Y  +619.956, Z    +0.000, E1   -63.110, E3 +232362.566}
SPL {X  -162.820, Y  +634.513, Z    +0.000, E1   -63.471, E3 +232375.332}
SPL {X  -162.820, Y  +648.936, Z    +0.000, E1   -63.278, E3 +232391.787}
SPL {X  -162.820, Y  +662.662, Z    +0.000, E1   -63.383, E3 +232405.279}
SPL {X  -162.819, Y  +673.983, Z    +0.000, E1   -63.398, E3 +232417.002}
SPL {X  -162.399, Y  +685.202, Z    +0.000, E1   -63.235, E3 +232429.996}
SPL {X  -161.289, Y  +695.772, Z    +0.000, E1   -63.167, E3 +232441.445}
SPL {X  -160.212, Y  +702.527, Z    +0.000, E1   -62.898, E3 +232450.426}
SPL {X  -158.647, Y  +710.128, Z    +0.000, E1   -62.776, E3 +232459.249}
SPL {X  -156.957, Y  +716.799, Z    +0.000, E1   -62.460, E3 +232468.367}
SPL {X  -154.447, Y  +725.041, Z    +0.000, E1   -62.170, E3 +232479.024}
SPL {X  -151.721, Y  +732.586, Z    +0.000, E1   -61.616, E3 +232490.274}
SPL {X  -149.420, Y  +738.185, Z    +0.000, E1   -61.282, E3 +232498.163}
SPL {X  -146.033, Y  +745.504, Z    +0.000, E1   -60.844, E3 +232508.430}
SPL {X  -142.518, Y  +752.234, Z    +0.000, E1   -60.144, E3 +232519.057}
SPL {X  -139.430, Y  +757.582, Z    +0.000, E1   -59.554, E3 +232527.589}
SPL {X  -134.550, Y  +765.187, Z    +0.000, E1   -59.954, E3 +232533.540}
SPL {X  -102.851, Y  +799.722, Z    +0.000, E1   -53.923, E3 +232624.032}
SPL {X  -101.618, Y  +800.716, Z    +0.000, E1   -52.212, E3 +232737.018}
ENDSPLINE

SPLINE
SPL {X  -141.567, Y  +753.931, Z    +0.000, E1   -42.659, E3 +232773.720}
SPL {X  -155.442, Y  +721.958, Z    +0.000, E1   -30.769, E3 +232780.626}
SPL {X  -161.417, Y  +694.832, Z    +0.000, E1   -16.464, E3 +232784.595}
SPL {X  -162.580, Y  +682.344, Z    +0.000, E1    -8.212, E3 +232784.802}
SPL {X  -162.811, Y  +675.182, Z    +0.000, E1    -3.078, E3 +232784.834}
SPL {X  -162.820, Y  +671.474, Z    +0.000, E1    -0.022, E3 +232784.304}
SPL {X  -162.820, Y  +668.525, Z    +0.000, E1    +3.543, E3 +232783.998}
SPL {X  -162.820, Y  +663.189, Z    +0.000, E1   +11.952, E3 +232783.987}
SPL {X  -162.820, Y  +655.445, Z    +0.000, E1   +24.952, E3 +232783.933}
SPL {X  -162.820, Y  +644.088, Z    +0.000, E1   +41.840, E3 +232784.070}
SPL {X  -162.820, Y  +632.645, Z    +0.000, E1   +53.114, E3 +232784.805}
SPL {X  -162.820, Y  +584.142, Z    +0.000, E1   +66.966, E3 +232800.148}
SPL {X  -162.820, Y  +471.906, Z    +0.000, E1   +66.781, E3 +232882.389}
ENDSPLINE

SPLINE
SPL {X  -162.820, Y  +475.237, Z    +0.000, E1   +64.883, E3 +232894.076}
ENDSPLINE

SPLINE
SPL {X  -162.820, Y  +462.171, Z    +0.000, E1   +64.935, E3 +232906.563}
SPL {X  -162.820, Y  +448.581, Z    +0.000, E1   +64.948, E3 +232919.574}
SPL {X  -162.820, Y  +437.579, Z    +0.000, E1   +64.893, E3 +232930.750}
SPL {X  -162.820, Y  +425.248, Z    +0.000, E1   +64.950, E3 +232942.337}
SPL {X  -162.820, Y  +417.868, Z    +0.000, E1   +64.478, E3 +232953.156}
ENDSPLINE

SPLINE
SPL {X  -162.820, Y  +442.889, Z    +0.000, E1   +58.918, E3 +232965.336}
ENDSPLINE

SPLINE
SPL {X  -162.820, Y  +428.091, Z    +0.000, E1   +59.583, E3 +232979.109}
SPL {X  -162.820, Y  +417.107, Z    +0.000, E1   +60.148, E3 +232988.510}
SPL {X  -162.820, Y  +398.797, Z    +0.000, E1   +61.348, E3 +233001.642}
SPL {X  -162.819, Y  +379.881, Z    +0.000, E1   +62.356, E3 +233015.472}
SPL {X  -162.597, Y  +371.985, Z    +0.000, E1   +62.420, E3 +233023.596}
SPL {X  -161.953, Y  +363.716, Z    +0.000, E1   +62.355, E3 +233033.053}
SPL {X  -160.528, Y  +353.277, Z    +0.000, E1   +62.144, E3 +233046.049}
SPL {X  -158.606, Y  +343.697, Z    +0.000, E1   +61.897, E3 +233057.953}
SPL {X  -156.311, Y  +334.925, Z    +0.000, E1   +61.505, E3 +233070.300}
SPL {X  -153.198, Y  +325.358, Z    +0.000, E1   +61.117, E3 +233082.992}
SPL {X  -151.022, Y  +319.651, Z    +0.000, E1   +60.776, E3 +233091.165}
SPL {X  -149.105, Y  +315.094, Z    +0.000, E1   +60.301, E3 +233098.918}
SPL {X  -146.196, Y  +308.826, Z    +0.000, E1   +59.961, E3 +233107.625}
SPL {X  -143.704, Y  +303.952, Z    +0.000, E1   +59.374, E3 +233115.982}
SPL {X  -140.940, Y  +298.976, Z    +0.000, E1   +59.075, E3 +233122.907}
SPL {X  -137.763, Y  +293.715, Z    +0.000, E1   +58.761, E3 +233130.013}
SPL {X  -129.725, Y  +282.103, Z    +0.000, E1   +61.069, E3 +233131.517}
SPL {X  -106.695, Y  +257.510, Z    +0.000, E1   +52.408, E3 +233232.239}
SPL {X  -104.122, Y  +255.325, Z    +0.000, E1   +51.312, E3 +233322.297}
ENDSPLINE

SPLINE
SPL {X  -140.007, Y  +297.383, Z    +0.000, E1   +42.766, E3 +233361.621}
SPL {X  -156.919, Y  +337.064, Z    +0.000, E1   +27.647, E3 +233367.772}
SPL {X  -161.737, Y  +361.753, Z    +0.000, E1   +14.421, E3 +233371.670}
SPL {X  -162.752, Y  +375.778, Z    +0.000, E1    +5.236, E3 +233371.862}
SPL {X  -162.820, Y  +381.939, Z    +0.000, E1    +0.593, E3 +233371.489}
SPL {X  -162.820, Y  +383.993, Z    +0.000, E1    -1.497, E3 +233371.062}
SPL {X  -162.820, Y  +387.367, Z    +0.000, E1    -6.003, E3 +233371.068}
SPL {X  -162.820, Y  +390.506, Z    +0.000, E1   -10.770, E3 +233370.811}
SPL {X  -162.820, Y  +394.643, Z    +0.000, E1   -17.317, E3 +233370.765}
SPL {X  -162.820, Y  +401.515, Z    +0.000, E1   -27.960, E3 +233371.585}
SPL {X  -162.820, Y  +412.105, Z    +0.000, E1   -42.847, E3 +233370.577}
SPL {X  -162.820, Y  +422.796, Z    +0.000, E1   -52.392, E3 +233371.797}
SPL {X  -162.820, Y  +474.423, Z    +0.000, E1   -65.078, E3 +233392.848}
SPL {X  -162.820, Y  +578.686, Z    +0.000, E1   -67.085, E3 +233462.013}
ENDSPLINE

SPLINE
SPL {X  -162.820, Y  +565.364, Z    +0.000, E1   -63.589, E3 +233476.013}
ENDSPLINE

SPLINE
SPL {X  -162.820, Y  +574.608, Z    +0.000, E1   -63.370, E3 +233487.272}
SPL {X  -162.820, Y  +584.314, Z    +0.000, E1   -63.342, E3 +233497.564}
SPL {X  -162.820, Y  +593.857, Z    +0.000, E1   -63.382, E3 +233507.266}
SPL {X  -162.820, Y  +602.272, Z    +0.000, E1   -63.279, E3 +233516.794}
SPL {X  -162.820, Y  +613.309, Z    +0.000, E1   -63.489, E3 +233526.793}
SPL {X  -162.820, Y  +627.013, Z    +0.000, E1   -63.389, E3 +233542.014}
SPL {X  -162.820, Y  +642.772, Z    +0.000, E1   -63.348, E3 +233558.672}
SPL {X  -162.820, Y  +651.969, Z    +0.000, E1   -63.137, E3 +233569.735}
SPL {X  -162.820, Y  +662.662, Z    +0.000, E1   -63.383, E3 +233579.192}
SPL {X  -162.819, Y  +673.983, Z    +0.000, E1   -63.398, E3 +233590.915}
SPL {X  -162.399, Y  +685.202, Z    +0.000, E1   -63.235, E3 +233603.909}
SPL {X  -161.289, Y  +695.772, Z    +0.000, E1   -63.167, E3 +233615.358}
SPL {X  -160.212, Y  +702.527, Z    +0.000, E1   -62.898, E3 +233624.339}
SPL {X  -158.647, Y  +710.128, Z    +0.000, E1   -62.776, E3 +233633.162}
SPL {X  -156.957, Y  +716.799, Z    +0.000, E1   -62.460, E3 +233642.280}
SPL {X  -155.130, Y  +722.947, Z    +0.000, E1   -62.207, E3 +233650.392}
SPL {X  -152.287, Y  +731.112, Z    +0.000, E1   -61.798, E3 +233661.668}
SPL {X  -149.420, Y  +738.185, Z    +0.000, E1   -61.282, E3 +233672.077}
SPL {X  -146.960, Y  +743.593, Z    +0.000, E1   -60.951, E3 +233679.620}
SPL {X  -143.277, Y  +750.844, Z    +0.000, E1   -60.348, E3 +233690.627}
SPL {X  -139.430, Y  +757.582, Z    +0.000, E1   -59.554, E3 +233701.502}
SPL {X  -134.550, Y  +765.187, Z    +0.000, E1   -59.954, E3 +233707.453}
SPL {X  -100.103, Y  +801.912, Z    +0.000, E1   -53.794, E3 +233805.503}
ENDSPLINE

SPLINE
SPL {X  -112.938, Y  +790.784, Z    +0.000, E1   -51.983, E3 +233941.025}
SPL {X  -141.567, Y  +753.931, Z    +0.000, E1   -42.659, E3 +233947.633}
SPL {X  -155.442, Y  +721.958, Z    +0.000, E1   -30.769, E3 +233954.539}
SPL {X  -161.417, Y  +694.832, Z    +0.000, E1   -16.464, E3 +233958.508}
SPL {X  -162.719, Y  +679.228, Z    +0.000, E1    -6.085, E3 +233958.832}
SPL {X  -162.820, Y  +673.638, Z    +0.000, E1    -1.806, E3 +233958.622}
SPL {X  -162.820, Y  +671.474, Z    +0.000, E1    -0.022, E3 +233958.217}
SPL {X  -162.820, Y  +668.525, Z    +0.000, E1    +3.543, E3 +233957.911}
SPL {X  -162.820, Y  +663.189, Z    +0.000, E1   +11.952, E3 +233957.900}
SPL {X  -162.820, Y  +657.986, Z    +0.000, E1   +20.997, E3 +233957.614}
SPL {X  -162.820, Y  +652.680, Z    +0.000, E1   +29.565, E3 +233958.099}
SPL {X  -162.820, Y  +644.088, Z    +0.000, E1   +41.840, E3 +233957.983}
SPL {X  -162.820, Y  +632.645, Z    +0.000, E1   +53.114, E3 +233958.718}
SPL {X  -162.820, Y  +584.142, Z    +0.000, E1   +66.966, E3 +233974.061}
SPL {X  -162.820, Y  +471.906, Z    +0.000, E1   +66.781, E3 +234056.302}
SPL {X  -162.820, Y  +470.218, Z    +0.000, E1   +64.979, E3 +234072.303}
SPL {X  -162.820, Y  +452.619, Z    +0.000, E1   +64.912, E3 +234089.981}
SPL {X  -162.820, Y  +437.579, Z    +0.000, E1   +64.893, E3 +234104.663}
SPL {X  -162.820, Y  +425.248, Z    +0.000, E1   +64.950, E3 +234116.250}
SPL {X  -162.820, Y  +417.868, Z    +0.000, E1   +64.478, E3 +234127.069}
ENDSPLINE

SPLINE
SPL {X  -162.820, Y  +442.889, Z    +0.000, E1   +58.918, E3 +234139.249}
ENDSPLINE

SPLINE
SPL {X  -162.820, Y  +428.091, Z    +0.000, E1   +59.583, E3 +234153.022}
SPL {X  -162.820, Y  +417.107, Z    +0.000, E1   +60.148, E3 +234162.423}
SPL {X  -162.820, Y  +398.797, Z    +0.000, E1   +61.348, E3 +234175.555}
SPL {X  -162.753, Y  +375.814, Z    +0.000, E1   +62.427, E3 +234193.478}
SPL {X  -161.572, Y  +360.382, Z    +0.000, E1   +62.315, E3 +234211.080}
SPL {X  -160.005, Y  +350.357, Z    +0.000, E1   +62.043, E3 +234223.644}
SPL {X  -158.606, Y  +343.697, Z    +0.000, E1   +61.897, E3 +234231.866}
SPL {X  -156.311, Y  +334.925, Z    +0.000, E1   +61.505, E3 +234244.213}
SPL {X  -153.198, Y  +325.358, Z    +0.000, E1   +61.117, E3 +234256.905}
SPL {X  -151.022, Y  +319.651, Z    +0.000, E1   +60.776, E3 +234265.078}
SPL {X  -149.105, Y  +315.094, Z    +0.000, E1   +60.301, E3 +234272.831}
SPL {X  -146.196, Y  +308.826, Z    +0.000, E1   +59.961, E3 +234281.538}
SPL {X  -143.704, Y  +303.952, Z    +0.000, E1   +59.374, E3 +234289.895}
SPL {X  -140.940, Y  +298.976, Z    +0.000, E1   +59.075, E3 +234296.820}
SPL {X  -137.763, Y  +293.715, Z    +0.000, E1   +58.761, E3 +234303.926}
SPL {X  -129.725, Y  +282.103, Z    +0.000, E1   +61.069, E3 +234305.430}
SPL {X  -106.695, Y  +257.510, Z    +0.000, E1   +52.408, E3 +234406.152}
SPL {X  -104.122, Y  +255.325, Z    +0.000, E1   +51.312, E3 +234496.210}
ENDSPLINE

SPLINE
SPL {X  -140.007, Y  +297.383, Z    +0.000, E1   +42.766, E3 +234535.534}
SPL {X  -155.551, Y  +332.393, Z    +0.000, E1   +29.794, E3 +234541.456}
SPL {X  -159.755, Y  +349.054, Z    +0.000, E1   +21.610, E3 +234543.329}
SPL {X  -162.078, Y  +364.978, Z    +0.000, E1   +12.369, E3 +234546.066}
SPL {X  -162.752, Y  +375.778, Z    +0.000, E1    +5.236, E3 +234545.775}
SPL {X  -162.820, Y  +381.939, Z    +0.000, E1    +0.593, E3 +234545.402}
SPL {X  -162.820, Y  +383.993, Z    +0.000, E1    -1.497, E3 +234544.975}
SPL {X  -162.820, Y  +388.628, Z    +0.000, E1    -7.678, E3 +234544.878}
SPL {X  -162.820, Y  +394.643, Z    +0.000, E1   -17.317, E3 +234544.678}
SPL {X  -162.820, Y  +401.515, Z    +0.000, E1   -27.960, E3 +234545.498}
SPL {X  -162.820, Y  +412.105, Z    +0.000, E1   -42.847, E3 +234544.490}
SPL {X  -162.820, Y  +422.796, Z    +0.000, E1   -52.392, E3 +234545.710}
SPL {X  -162.820, Y  +474.423, Z    +0.000, E1   -65.078, E3 +234566.761}
SPL {X  -162.820, Y  +578.686, Z    +0.000, E1   -67.085, E3 +234635.926}
ENDSPLINE

SPLINE
SPL {X  -162.820, Y  +565.364, Z    +0.000, E1   -63.589, E3 +234649.926}
ENDSPLINE

SPLINE
SPL {X  -162.820, Y  +574.608, Z    +0.000, E1   -63.370, E3 +234661.185}
SPL {X  -162.820, Y  +584.314, Z    +0.000, E1   -63.342, E3 +234671.477}
SPL {X  -162.820, Y  +593.857, Z    +0.000, E1   -63.382, E3 +234681.179}
SPL {X  -162.820, Y  +602.272, Z    +0.000, E1   -63.279, E3 +234690.707}
SPL {X  -162.820, Y  +613.309, Z    +0.000, E1   -63.489, E3 +234700.706}
SPL {X  -162.820, Y  +619.956, Z    +0.000, E1   -63.110, E3 +234710.392}
SPL {X  -162.820, Y  +631.846, Z    +0.000, E1   -63.529, E3 +234719.783}
SPL {X  -162.820, Y  +642.772, Z    +0.000, E1   -63.348, E3 +234732.585}
SPL {X  -162.820, Y  +658.642, Z    +0.000, E1   -63.324, E3 +234749.500}
SPL {X  -162.819, Y  +673.983, Z    +0.000, E1   -63.398, E3 +234764.828}
SPL {X  -162.617, Y  +681.634, Z    +0.000, E1   -63.169, E3 +234774.450}
SPL {X  -161.618, Y  +693.246, Z    +0.000, E1   -63.233, E3 +234786.308}
SPL {X  -160.212, Y  +702.527, Z    +0.000, E1   -62.898, E3 +234798.252}
SPL {X  -158.647, Y  +710.128, Z    +0.000, E1   -62.776, E3 +234807.075}
SPL {X  -156.957, Y  +716.799, Z    +0.000, E1   -62.460, E3 +234816.193}
SPL {X  -154.447, Y  +725.041, Z    +0.000, E1   -62.170, E3 +234826.850}
SPL {X  -151.721, Y  +732.586, Z    +0.000, E1   -61.616, E3 +234838.100}
SPL {X  -149.420, Y  +738.185, Z    +0.000, E1   -61.282, E3 +234845.990}
SPL {X  -146.033, Y  +745.504, Z    +0.000, E1   -60.844, E3 +234856.256}
SPL {X  -142.518, Y  +752.234, Z    +0.000, E1   -60.144, E3 +234866.883}
SPL {X  -139.430, Y  +757.582, Z    +0.000, E1   -59.554, E3 +234875.415}
SPL {X  -134.550, Y  +765.187, Z    +0.000, E1   -59.954, E3 +234881.366}
SPL {X  -100.103, Y  +801.912, Z    +0.000, E1   -53.794, E3 +234979.416}
ENDSPLINE

SPLINE
SPL {X  -112.938, Y  +790.784, Z    +0.000, E1   -51.983, E3 +235114.938}
SPL {X  -141.567, Y  +753.931, Z    +0.000, E1   -42.659, E3 +235121.546}
SPL {X  -155.442, Y  +721.958, Z    +0.000, E1   -30.769, E3 +235128.452}
SPL {X  -161.417, Y  +694.832, Z    +0.000, E1   -16.464, E3 +235132.421}
SPL {X  -162.580, Y  +682.344, Z    +0.000, E1    -8.212, E3 +235132.628}
SPL {X  -162.811, Y  +675.182, Z    +0.000, E1    -3.078, E3 +235132.660}
SPL {X  -162.820, Y  +670.948, Z    +0.000, E1    +0.412, E3 +235132.059}
SPL {X  -162.820, Y  +667.375, Z    +0.000, E1    +5.386, E3 +235131.749}
SPL {X  -162.820, Y  +663.189, Z    +0.000, E1   +11.952, E3 +235131.813}
SPL {X  -162.820, Y  +655.445, Z    +0.000, E1   +24.952, E3 +235131.759}
SPL {X  -162.820, Y  +644.088, Z    +0.000, E1   +41.840, E3 +235131.896}
SPL {X  -162.820, Y  +632.645, Z    +0.000, E1   +53.114, E3 +235132.631}
SPL {X  -162.820, Y  +584.142, Z    +0.000, E1   +66.966, E3 +235147.974}
SPL {X  -162.820, Y  +471.906, Z    +0.000, E1   +66.781, E3 +235230.216}
SPL {X  -162.820, Y  +470.218, Z    +0.000, E1   +64.979, E3 +235246.216}
SPL {X  -162.820, Y  +452.619, Z    +0.000, E1   +64.912, E3 +235263.894}
SPL {X  -162.820, Y  +437.579, Z    +0.000, E1   +64.893, E3 +235278.576}
SPL {X  -162.820, Y  +425.248, Z    +0.000, E1   +64.950, E3 +235290.163}
SPL {X  -162.820, Y  +417.868, Z    +0.000, E1   +64.478, E3 +235300.982}
ENDSPLINE

SPLINE
SPL {X  -162.820, Y  +442.889, Z    +0.000, E1   +58.918, E3 +235313.162}
ENDSPLINE

SPLINE
SPL {X  -162.820, Y  +428.091, Z    +0.000, E1   +59.583, E3 +235326.935}
SPL {X  -162.820, Y  +417.107, Z    +0.000, E1   +60.148, E3 +235336.336}
SPL {X  -162.820, Y  +398.797, Z    +0.000, E1   +61.348, E3 +235349.469}
SPL {X  -162.753, Y  +375.814, Z    +0.000, E1   +62.427, E3 +235367.391}
SPL {X  -161.572, Y  +360.382, Z    +0.000, E1   +62.315, E3 +235384.993}
SPL {X  -160.005, Y  +350.357, Z    +0.000, E1   +62.043, E3 +235397.557}
SPL {X  -158.606, Y  +343.697, Z    +0.000, E1   +61.897, E3 +235405.779}
SPL {X  -156.311, Y  +334.925, Z    +0.000, E1   +61.505, E3 +235418.126}
SPL {X  -153.198, Y  +325.358, Z    +0.000, E1   +61.117, E3 +235430.818}
SPL {X  -151.022, Y  +319.651, Z    +0.000, E1   +60.776, E3 +235438.991}
SPL {X  -149.105, Y  +315.094, Z    +0.000, E1   +60.301, E3 +235446.744}
SPL {X  -146.196, Y  +308.826, Z    +0.000, E1   +59.961, E3 +235455.451}
SPL {X  -143.704, Y  +303.952, Z    +0.000, E1   +59.374, E3 +235463.808}
SPL {X  -140.940, Y  +298.976, Z    +0.000, E1   +59.075, E3 +235470.733}
SPL {X  -137.763, Y  +293.715, Z    +0.000, E1   +58.761, E3 +235477.839}
SPL {X  -129.725, Y  +282.103, Z    +0.000, E1   +61.069, E3 +235479.343}
SPL {X  -106.695, Y  +257.510, Z    +0.000, E1   +52.408, E3 +235580.065}
SPL {X  -104.122, Y  +255.325, Z    +0.000, E1   +51.312, E3 +235670.123}
ENDSPLINE

SPLINE
SPL {X  -140.007, Y  +297.383, Z    +0.000, E1   +42.766, E3 +235709.448}
SPL {X  -156.919, Y  +337.064, Z    +0.000, E1   +27.647, E3 +235715.598}
SPL {X  -161.737, Y  +361.753, Z    +0.000, E1   +14.421, E3 +235719.496}
SPL {X  -162.752, Y  +375.778, Z    +0.000, E1    +5.236, E3 +235719.688}
SPL {X  -162.820, Y  +381.939, Z    +0.000, E1    +0.593, E3 +235719.315}
SPL {X  -162.820, Y  +383.993, Z    +0.000, E1    -1.497, E3 +235718.888}
SPL {X  -162.820, Y  +388.628, Z    +0.000, E1    -7.678, E3 +235718.791}
SPL {X  -162.820, Y  +394.643, Z    +0.000, E1   -17.317, E3 +235718.591}
SPL {X  -162.820, Y  +401.515, Z    +0.000, E1   -27.960, E3 +235719.411}
SPL {X  -162.820, Y  +412.105, Z    +0.000, E1   -42.847, E3 +235718.403}
SPL {X  -162.820, Y  +422.796, Z    +0.000, E1   -52.392, E3 +235719.623}
SPL {X  -162.820, Y  +474.423, Z    +0.000, E1   -65.078, E3 +235740.674}
SPL {X  -162.820, Y  +578.686, Z    +0.000, E1   -67.085, E3 +235809.839}
ENDSPLINE

SPLINE
SPL {X  -162.820, Y  +565.364, Z    +0.000, E1   -63.589, E3 +235823.839}
ENDSPLINE

SPLINE
SPL {X  -162.820, Y  +574.608, Z    +0.000, E1   -63.370, E3 +235835.098}
SPL {X  -162.820, Y  +584.314, Z    +0.000, E1   -63.342, E3 +235845.390}
SPL {X  -162.820, Y  +593.857, Z    +0.000, E1   -63.382, E3 +235855.092}
SPL {X  -162.820, Y  +602.272, Z    +0.000, E1   -63.279, E3 +235864.620}
SPL {X  -162.820, Y  +613.309, Z    +0.000, E1   -63.489, E3 +235874.619}
SPL {X  -162.820, Y  +619.956, Z    +0.000, E1   -63.110, E3 +235884.305}
SPL {X  -162.820, Y  +631.846, Z    +0.000, E1   -63.529, E3 +235893.696}
SPL {X  -162.820, Y  +642.772, Z    +0.000, E1   -63.348, E3 +235906.498}
SPL {X  -162.820, Y  +658.642, Z    +0.000, E1   -63.324, E3 +235923.413}
SPL {X  -162.819, Y  +673.983, Z    +0.000, E1   -63.398, E3 +235938.741}
SPL {X  -162.399, Y  +685.202, Z    +0.000, E1   -63.235, E3 +235951.735}
SPL {X  -161.289, Y  +695.772, Z    +0.000, E1   -63.167, E3 +235963.185}
SPL {X  -160.212, Y  +702.527, Z    +0.000, E1   -62.898, E3 +235972.165}
SPL {X  -158.647, Y  +710.128, Z    +0.000, E1   -62.776, E3 +235980.988}
SPL {X  -156.957, Y  +716.799, Z    +0.000, E1   -62.460, E3 +235990.106}
SPL {X  -154.447, Y  +725.041, Z    +0.000, E1   -62.170, E3 +236000.763}
SPL {X  -151.721, Y  +732.586, Z    +0.000, E1   -61.616, E3 +236012.013}
SPL {X  -149.420, Y  +738.185, Z    +0.000, E1   -61.282, E3 +236019.903}
SPL {X  -146.960, Y  +743.593, Z    +0.000, E1   -60.951, E3 +236027.446}
SPL {X  -143.277, Y  +750.844, Z    +0.000, E1   -60.348, E3 +236038.453}
SPL {X  -139.430, Y  +757.582, Z    +0.000, E1   -59.554, E3 +236049.328}
SPL {X  -134.550, Y  +765.187, Z    +0.000, E1   -59.954, E3 +236055.279}
SPL {X  -100.103, Y  +801.912, Z    +0.000, E1   -53.794, E3 +236153.329}
ENDSPLINE

SPLINE
SPL {X  -112.938, Y  +790.784, Z    +0.000, E1   -51.983, E3 +236288.851}
SPL {X  -141.567, Y  +753.931, Z    +0.000, E1   -42.659, E3 +236295.459}
SPL {X  -155.442, Y  +721.958, Z    +0.000, E1   -30.769, E3 +236302.365}
SPL {X  -161.417, Y  +694.832, Z    +0.000, E1   -16.464, E3 +236306.334}
SPL {X  -162.719, Y  +679.228, Z    +0.000, E1    -6.085, E3 +236306.658}
SPL {X  -162.820, Y  +673.638, Z    +0.000, E1    -1.806, E3 +236306.448}
SPL {X  -162.820, Y  +670.948, Z    +0.000, E1    +0.412, E3 +236305.972}
SPL {X  -162.820, Y  +667.375, Z    +0.000, E1    +5.386, E3 +236305.662}
SPL {X  -162.820, Y  +663.189, Z    +0.000, E1   +11.952, E3 +236305.726}
SPL {X  -162.820, Y  +655.445, Z    +0.000, E1   +24.952, E3 +236305.672}
SPL {X  -162.820, Y  +644.088, Z    +0.000, E1   +41.840, E3 +236305.809}
SPL {X  -162.820, Y  +632.645, Z    +0.000, E1   +53.114, E3 +236306.544}
SPL {X  -162.820, Y  +584.142, Z    +0.000, E1   +66.966, E3 +236321.887}
SPL {X  -162.820, Y  +471.906, Z    +0.000, E1   +66.781, E3 +236404.129}
SPL {X  -162.820, Y  +470.218, Z    +0.000, E1   +64.979, E3 +236420.129}
SPL {X  -162.820, Y  +452.619, Z    +0.000, E1   +64.912, E3 +236437.807}
SPL {X  -162.820, Y  +437.579, Z    +0.000, E1   +64.893, E3 +236452.489}
SPL {X  -162.820, Y  +425.248, Z    +0.000, E1   +64.950, E3 +236464.076}
SPL {X  -162.820, Y  +417.868, Z    +0.000, E1   +64.478, E3 +236474.895}
ENDSPLINE

SPLINE
SPL {X  -162.820, Y  +447.149, Z    +0.000, E1   +58.721, E3 +236482.891}
ENDSPLINE

SPLINE
SPL {X  -162.820, Y  +431.862, Z    +0.000, E1   +59.419, E3 +236497.439}
SPL {X  -162.820, Y  +417.107, Z    +0.000, E1   +60.148, E3 +236510.249}
SPL {X  -162.820, Y  +398.797, Z    +0.000, E1   +61.348, E3 +236523.382}
SPL {X  -162.753, Y  +375.814, Z    +0.000, E1   +62.427, E3 +236541.304}
SPL {X  -161.953, Y  +363.716, Z    +0.000, E1   +62.355, E3 +236554.792}
SPL {X  -160.528, Y  +353.277, Z    +0.000, E1   +62.144, E3 +236567.788}
SPL {X  -157.973, Y  +341.066, Z    +0.000, E1   +61.800, E3 +236583.387}
SPL {X  -155.627, Y  +332.640, Z    +0.000, E1   +61.354, E3 +236595.301}
SPL {X  -153.198, Y  +325.358, Z    +0.000, E1   +61.117, E3 +236604.731}
SPL {X  -151.022, Y  +319.651, Z    +0.000, E1   +60.776, E3 +236612.904}
SPL {X  -149.105, Y  +315.094, Z    +0.000, E1   +60.301, E3 +236620.657}
SPL {X  -146.196, Y  +308.826, Z    +0.000, E1   +59.961, E3 +236629.364}
SPL {X  -143.704, Y  +303.952, Z    +0.000, E1   +59.374, E3 +236637.721}
SPL {X  -140.940, Y  +298.976, Z    +0.000, E1   +59.075, E3 +236644.646}
SPL {X  -137.763, Y  +293.715, Z    +0.000, E1   +58.761, E3 +236651.752}
SPL {X  -129.725, Y  +282.103, Z    +0.000, E1   +61.069, E3 +236653.256}
SPL {X  -106.695, Y  +257.510, Z    +0.000, E1   +52.408, E3 +236753.978}
SPL {X  -104.122, Y  +255.325, Z    +0.000, E1   +51.312, E3 +236844.036}
ENDSPLINE

SPLINE
SPL {X  -140.007, Y  +297.383, Z    +0.000, E1   +42.766, E3 +236883.361}
SPL {X  -156.919, Y  +337.064, Z    +0.000, E1   +27.647, E3 +236889.512}
SPL {X  -161.737, Y  +361.753, Z    +0.000, E1   +14.421, E3 +236893.409}
SPL {X  -162.752, Y  +375.778, Z    +0.000, E1    +5.236, E3 +236893.601}
SPL {X  -162.820, Y  +382.443, Z    +0.000, E1    +0.212, E3 +236893.081}
SPL {X  -162.820, Y  +386.214, Z    +0.000, E1    -4.241, E3 +236892.783}
SPL {X  -162.820, Y  +390.506, Z    +0.000, E1   -10.770, E3 +236892.550}
SPL {X  -162.820, Y  +394.643, Z    +0.000, E1   -17.317, E3 +236892.504}
SPL {X  -162.820, Y  +401.515, Z    +0.000, E1   -27.960, E3 +236893.324}
SPL {X  -162.820, Y  +412.105, Z    +0.000, E1   -42.847, E3 +236892.316}
SPL {X  -162.820, Y  +422.796, Z    +0.000, E1   -52.392, E3 +236893.536}
SPL {X  -162.820, Y  +474.423, Z    +0.000, E1   -65.078, E3 +236914.587}
SPL {X  -162.820, Y  +578.686, Z    +0.000, E1   -67.085, E3 +236983.752}
ENDSPLINE

SPLINE
SPL {X  -162.820, Y  +565.364, Z    +0.000, E1   -63.589, E3 +236997.752}
ENDSPLINE

SPLINE
SPL {X  -162.820, Y  +574.608, Z    +0.000, E1   -63.370, E3 +237009.011}
SPL {X  -162.820, Y  +584.314, Z    +0.000, E1   -63.342, E3 +237019.303}
SPL {X  -162.820, Y  +593.857, Z    +0.000, E1   -63.382, E3 +237029.005}
SPL {X  -162.820, Y  +602.272, Z    +0.000, E1   -63.279, E3 +237038.533}
SPL {X  -162.820, Y  +613.309, Z    +0.000, E1   -63.489, E3 +237048.532}
SPL {X  -162.820, Y  +627.013, Z    +0.000, E1   -63.389, E3 +237063.753}
SPL {X  -162.820, Y  +642.772, Z    +0.000, E1   -63.348, E3 +237080.411}
SPL {X  -162.820, Y  +658.642, Z    +0.000, E1   -63.324, E3 +237097.326}
SPL {X  -162.819, Y  +673.983, Z    +0.000, E1   -63.398, E3 +237112.654}
SPL {X  -162.617, Y  +681.634, Z    +0.000, E1   -63.169, E3 +237122.276}
SPL {X  -161.618, Y  +693.246, Z    +0.000, E1   -63.233, E3 +237134.134}
SPL {X  -160.212, Y  +702.527, Z    +0.000, E1   -62.898, E3 +237146.078}
SPL {X  -158.647, Y  +710.128, Z    +0.000, E1   -62.776, E3 +237154.901}
SPL {X  -156.957, Y  +716.799, Z    +0.000, E1   -62.460, E3 +237164.019}
SPL {X  -155.130, Y  +722.947, Z    +0.000, E1   -62.207, E3 +237172.132}
SPL {X  -152.287, Y  +731.112, Z    +0.000, E1   -61.798, E3 +237183.407}
SPL {X  -149.420, Y  +738.185, Z    +0.000, E1   -61.282, E3 +237193.816}
SPL {X  -146.033, Y  +745.504, Z    +0.000, E1   -60.844, E3 +237204.083}
SPL {X  -142.518, Y  +752.234, Z    +0.000, E1   -60.144, E3 +237214.709}
SPL {X  -139.430, Y  +757.582, Z    +0.000, E1   -59.554, E3 +237223.241}
SPL {X  -134.550, Y  +765.187, Z    +0.000, E1   -59.954, E3 +237229.192}
SPL {X  -100.103, Y  +801.912, Z    +0.000, E1   -53.794, E3 +237327.242}
ENDSPLINE

SPLINE
SPL {X  -112.938, Y  +790.784, Z    +0.000, E1   -51.983, E3 +237462.764}
SPL {X  -141.567, Y  +753.931, Z    +0.000, E1   -42.659, E3 +237469.372}
SPL {X  -155.442, Y  +721.958, Z    +0.000, E1   -30.769, E3 +237476.278}
SPL {X  -161.417, Y  +694.832, Z    +0.000, E1   -16.464, E3 +237480.247}
SPL {X  -162.719, Y  +679.228, Z    +0.000, E1    -6.085, E3 +237480.571}
SPL {X  -162.820, Y  +673.638, Z    +0.000, E1    -1.806, E3 +237480.361}
SPL {X  -162.820, Y  +670.948, Z    +0.000, E1    +0.412, E3 +237479.885}
SPL {X  -162.820, Y  +667.375, Z    +0.000, E1    +5.386, E3 +237479.575}
SPL {X  -162.820, Y  +663.189, Z    +0.000, E1   +11.952, E3 +237479.639}
SPL {X  -162.820, Y  +655.445, Z    +0.000, E1   +24.952, E3 +237479.585}
SPL {X  -162.820, Y  +644.088, Z    +0.000, E1   +41.840, E3 +237479.722}
SPL {X  -162.820, Y  +632.645, Z    +0.000, E1   +53.114, E3 +237480.457}
SPL {X  -162.820, Y  +584.142, Z    +0.000, E1   +66.966, E3 +237495.800}
SPL {X  -162.820, Y  +466.182, Z    +0.000, E1   +68.456, E3 +237569.571}
ENDSPLINE

SPLINE
SPL {X  -162.820, Y  +475.083, Z    +0.000, E1   +65.244, E3 +237587.271}
ENDSPLINE

SPLINE
SPL {X  -162.820, Y  +465.389, Z    +0.000, E1   +65.015, E3 +237598.288}
SPL {X  -162.820, Y  +452.619, Z    +0.000, E1   +64.912, E3 +237611.720}
SPL {X  -162.820, Y  +437.579, Z    +0.000, E1   +64.893, E3 +237626.402}
SPL {X  -162.820, Y  +425.248, Z    +0.000, E1   +64.950, E3 +237637.989}
SPL {X  -162.820, Y  +417.868, Z    +0.000, E1   +64.478, E3 +237648.808}
ENDSPLINE

SPLINE
SPL {X  -162.820, Y  +442.889, Z    +0.000, E1   +58.918, E3 +237660.988}
ENDSPLINE

SPLINE
SPL {X  -162.820, Y  +428.091, Z    +0.000, E1   +59.583, E3 +237674.761}
SPL {X  -162.820, Y  +417.107, Z    +0.000, E1   +60.148, E3 +237684.162}
SPL {X  -162.820, Y  +398.797, Z    +0.000, E1   +61.348, E3 +237697.295}
SPL {X  -162.819, Y  +379.881, Z    +0.000, E1   +62.356, E3 +237711.125}
SPL {X  -162.597, Y  +371.985, Z    +0.000, E1   +62.420, E3 +237719.248}
SPL {X  -161.953, Y  +363.716, Z    +0.000, E1   +62.355, E3 +237728.705}
SPL {X  -160.528, Y  +353.277, Z    +0.000, E1   +62.144, E3 +237741.701}
SPL {X  -158.606, Y  +343.697, Z    +0.000, E1   +61.897, E3 +237753.606}
SPL {X  -156.311, Y  +334.925, Z    +0.000, E1   +61.505, E3 +237765.952}
SPL {X  -153.198, Y  +325.358, Z    +0.000, E1   +61.117, E3 +237778.644}
SPL {X  -151.022, Y  +319.651, Z    +0.000, E1   +60.776, E3 +237786.817}
SPL {X  -149.105, Y  +315.094, Z    +0.000, E1   +60.301, E3 +237794.570}
SPL {X  -146.196, Y  +308.826, Z    +0.000, E1   +59.961, E3 +237803.277}
SPL {X  -143.704, Y  +303.952, Z    +0.000, E1   +59.374, E3 +237811.634}
SPL {X  -140.940, Y  +298.976, Z    +0.000, E1   +59.075, E3 +237818.559}
SPL {X  -137.763, Y  +293.715, Z    +0.000, E1   +58.761, E3 +237825.665}
SPL {X  -129.725, Y  +282.103, Z    +0.000, E1   +61.069, E3 +237827.169}
SPL {X  -106.695, Y  +257.510, Z    +0.000, E1   +52.408, E3 +237927.891}
SPL {X  -104.122, Y  +255.325, Z    +0.000, E1   +51.312, E3 +238017.949}
ENDSPLINE

SPLINE
SPL {X  -140.007, Y  +297.383, Z    +0.000, E1   +42.766, E3 +238057.274}
SPL {X  -156.919, Y  +337.064, Z    +0.000, E1   +27.647, E3 +238063.425}
SPL {X  -160.736, Y  +354.534, Z    +0.000, E1   +18.553, E3 +238066.120}
SPL {X  -162.078, Y  +364.978, Z    +0.000, E1   +12.369, E3 +238067.805}
SPL {X  -162.656, Y  +373.196, Z    +0.000, E1    +6.960, E3 +238067.300}
SPL {X  -162.819, Y  +379.805, Z    +0.000, E1    +2.285, E3 +238067.424}
SPL {X  -162.820, Y  +382.398, Z    +0.000, E1    +0.126, E3 +238067.084}
SPL {X  -162.820, Y  +383.993, Z    +0.000, E1    -1.497, E3 +238066.714}
SPL {X  -162.820, Y  +387.367, Z    +0.000, E1    -6.003, E3 +238066.720}
SPL {X  -162.820, Y  +390.506, Z    +0.000, E1   -10.770, E3 +238066.463}
SPL {X  -162.820, Y  +394.643, Z    +0.000, E1   -17.317, E3 +238066.417}
SPL {X  -162.820, Y  +401.515, Z    +0.000, E1   -27.960, E3 +238067.237}
SPL {X  -162.820, Y  +412.105, Z    +0.000, E1   -42.847, E3 +238066.229}
SPL {X  -162.820, Y  +422.796, Z    +0.000, E1   -52.392, E3 +238067.450}
SPL {X  -162.820, Y  +474.423, Z    +0.000, E1   -65.078, E3 +238088.500}
SPL {X  -162.820, Y  +578.686, Z    +0.000, E1   -67.085, E3 +238157.665}
ENDSPLINE

SPLINE
SPL {X  -162.820, Y  +565.364, Z    +0.000, E1   -63.589, E3 +238171.665}
ENDSPLINE

SPLINE
SPL {X  -162.820, Y  +574.608, Z    +0.000, E1   -63.370, E3 +238182.924}
SPL {X  -162.820, Y  +584.314, Z    +0.000, E1   -63.342, E3 +238193.216}
SPL {X  -162.820, Y  +593.857, Z    +0.000, E1   -63.382, E3 +238202.918}
SPL {X  -162.820, Y  +602.272, Z    +0.000, E1   -63.279, E3 +238212.446}
SPL {X  -162.820, Y  +613.309, Z    +0.000, E1   -63.489, E3 +238222.445}
SPL {X  -162.820, Y  +619.956, Z    +0.000, E1   -63.110, E3 +238232.131}
SPL {X  -162.820, Y  +634.513, Z    +0.000, E1   -63.471, E3 +238244.897}
SPL {X  -162.820, Y  +648.936, Z    +0.000, E1   -63.278, E3 +238261.352}
SPL {X  -162.820, Y  +662.662, Z    +0.000, E1   -63.383, E3 +238274.844}
SPL {X  -162.819, Y  +673.983, Z    +0.000, E1   -63.398, E3 +238286.567}
SPL {X  -162.399, Y  +685.202, Z    +0.000, E1   -63.235, E3 +238299.561}
SPL {X  -161.289, Y  +695.772, Z    +0.000, E1   -63.167, E3 +238311.011}
SPL {X  -160.212, Y  +702.527, Z    +0.000, E1   -62.898, E3 +238319.991}
SPL {X  -158.647, Y  +710.128, Z    +0.000, E1   -62.776, E3 +238328.814}
SPL {X  -156.957, Y  +716.799, Z    +0.000, E1   -62.460, E3 +238337.932}
SPL {X  -154.447, Y  +725.041, Z    +0.000, E1   -62.170, E3 +238348.589}
SPL {X  -151.721, Y  +732.586, Z    +0.000, E1   -61.616, E3 +238359.839}
SPL {X  -149.420, Y  +738.185, Z    +0.000, E1   -61.282, E3 +238367.729}
SPL {X  -146.960, Y  +743.593, Z    +0.000, E1   -60.951, E3 +238375.273}
SPL {X  -143.277, Y  +750.844, Z    +0.000, E1   -60.348, E3 +238386.279}
SPL {X  -139.430, Y  +757.582, Z    +0.000, E1   -59.554, E3 +238397.154}
SPL {X  -134.550, Y  +765.187, Z    +0.000, E1   -59.954, E3 +238403.105}
SPL {X  -100.103, Y  +801.912, Z    +0.000, E1   -53.794, E3 +238501.155}
ENDSPLINE

SPLINE
SPL {X  -112.938, Y  +790.784, Z    +0.000, E1   -51.983, E3 +238636.677}
SPL {X  -145.058, Y  +747.450, Z    +0.000, E1   -40.634, E3 +238644.787}
SPL {X  -158.857, Y  +709.206, Z    +0.000, E1   -24.633, E3 +238652.756}
SPL {X  -161.919, Y  +690.607, Z    +0.000, E1   -13.733, E3 +238654.235}
SPL {X  -162.719, Y  +679.228, Z    +0.000, E1    -6.085, E3 +238654.484}
SPL {X  -162.820, Y  +671.750, Z    +0.000, E1    -0.355, E3 +238653.921}
SPL {X  -162.820, Y  +669.853, Z    +0.000, E1    +1.938, E3 +238653.651}
SPL {X  -162.820, Y  +667.375, Z    +0.000, E1    +5.386, E3 +238653.488}
SPL {X  -162.820, Y  +663.189, Z    +0.000, E1   +11.952, E3 +238653.552}
SPL {X  -162.820, Y  +657.986, Z    +0.000, E1   +20.997, E3 +238653.266}
SPL {X  -162.820, Y  +650.033, Z    +0.000, E1   +33.465, E3 +238653.736}
SPL {X  -162.820, Y  +635.632, Z    +0.000, E1   +50.654, E3 +238654.060}
SPL {X  -162.820, Y  +584.142, Z    +0.000, E1   +66.966, E3 +238669.713}
SPL {X  -162.820, Y  +466.182, Z    +0.000, E1   +68.456, E3 +238743.484}
ENDSPLINE

SPLINE
SPL {X  -162.820, Y  +475.083, Z    +0.000, E1   +65.244, E3 +238761.184}
ENDSPLINE

SPLINE
SPL {X  -162.820, Y  +465.389, Z    +0.000, E1   +65.015, E3 +238772.201}
SPL {X  -162.820, Y  +452.619, Z    +0.000, E1   +64.912, E3 +238785.633}
SPL {X  -162.820, Y  +437.579, Z    +0.000, E1   +64.893, E3 +238800.315}
SPL {X  -162.820, Y  +425.248, Z    +0.000, E1   +64.950, E3 +238811.903}
SPL {X  -162.820, Y  +417.868, Z    +0.000, E1   +64.478, E3 +238822.721}
ENDSPLINE

SPLINE
SPL {X  -162.820, Y  +442.889, Z    +0.000, E1   +58.918, E3 +238834.901}
ENDSPLINE

SPLINE
SPL {X  -162.820, Y  +428.091, Z    +0.000, E1   +59.583, E3 +238848.674}
SPL {X  -162.820, Y  +417.107, Z    +0.000, E1   +60.148, E3 +238858.075}
SPL {X  -162.820, Y  +398.797, Z    +0.000, E1   +61.348, E3 +238871.208}
SPL {X  -162.819, Y  +379.860, Z    +0.000, E1   +62.359, E3 +238885.037}
SPL {X  -162.598, Y  +372.005, Z    +0.000, E1   +62.416, E3 +238893.161}
SPL {X  -161.953, Y  +363.716, Z    +0.000, E1   +62.355, E3 +238902.618}
SPL {X  -160.528, Y  +353.277, Z    +0.000, E1   +62.144, E3 +238915.614}
SPL {X  -157.973, Y  +341.066, Z    +0.000, E1   +61.800, E3 +238931.213}
SPL {X  -155.627, Y  +332.640, Z    +0.000, E1   +61.354, E3 +238943.127}
SPL {X  -153.198, Y  +325.358, Z    +0.000, E1   +61.117, E3 +238952.557}
SPL {X  -151.022, Y  +319.651, Z    +0.000, E1   +60.776, E3 +238960.730}
SPL {X  -149.105, Y  +315.094, Z    +0.000, E1   +60.301, E3 +238968.483}
SPL {X  -146.196, Y  +308.826, Z    +0.000, E1   +59.961, E3 +238977.190}
SPL {X  -143.704, Y  +303.952, Z    +0.000, E1   +59.374, E3 +238985.547}
SPL {X  -140.940, Y  +298.976, Z    +0.000, E1   +59.075, E3 +238992.472}
SPL {X  -137.763, Y  +293.715, Z    +0.000, E1   +58.761, E3 +238999.579}
SPL {X  -129.725, Y  +282.103, Z    +0.000, E1   +61.069, E3 +239001.082}
SPL {X  -106.695, Y  +257.510, Z    +0.000, E1   +52.408, E3 +239101.804}
SPL {X  -104.122, Y  +255.325, Z    +0.000, E1   +51.312, E3 +239191.862}
ENDSPLINE

